// TwinCAT 3 PLC project Anthem
// ProgramVersion: 3.1.4023.0
// libraries:
//   Tc2_ModbusRTU, * (Beckhoff Automation GmbH)
//   Tc2_Standard, * (Beckhoff Automation GmbH)
//   Tc2_System, * (Beckhoff Automation GmbH)
//   Tc2_Utilities, * (Beckhoff Automation GmbH)
//   Tc3_Module, * (Beckhoff Automation GmbH)
// project tree:
//   / AnalogScaling.TcPOU, PlcTask.TcTTO
//   DUTs/ Block.TcDUT, EachRecipeStep.TcDUT, IndividualProcess.TcDUT, PhysicalIO.TcDUT, Properties.TcDUT, Pump.TcDUT, Reactor.TcDUT, Recipe.TcDUT, Valve.TcDUT, Vessel.TcDUT, VFD.TcDUT
//   GVLs/ IO.TcGVL, RecipeTags.TcGVL
//   Helpers/Assigner/ FB_Assigner.TcPOU, FB_TagAssignment.TcPOU, I_TagAssignment.TcIO
//   Helpers/ fbSimulator.TcPOU, FB_Scaling.TcPOU, MessageProvider.TcPOU, RecipeCommHandler.TcPOU
//   Helpers/RemainingTimeCalculator/ FBRemTimeCalc.TcPOU
//   Helpers/ShutDown/ FB_Shutdown.TcPOU, I_ShutDown.TcIO
//   Helpers/StirControl/ FbStirControl.TcPOU, IStirControl.TcIO
//   Helpers/VesselSelection/ FBSelection.TcPOU, ISelection.TcIO
//   ManualControl/ FB_ManualControl.TcPOU, I_ManualControl.TcIO
//   ManualControl/ManualImplementation/ FB_ManualImplementation.TcPOU, I_ManualImplementation.TcIO
//   Manualmplementation/ FB_ManualImplementation_1.TcPOU, I_ManualImplementation_1.TcIO
//   Manualmplementation/ManualControl/ FB_ManualControl_1.TcPOU, I_ManualControl_1.TcIO
//   POUs/ AnalogScaling_1.TcPOU, MAIN.TcPOU, Modbus.TcPOU
//   RecipeControl/ ClearRecipe.TcPOU, RecipeControl.TcPOU
//   RecipeControl/RecipeBlocks/Drain/ Drain.TcPOU
//   RecipeControl/RecipeBlocks/Flush/ FbFlush.TcPOU, IFlush.TcIO
//   RecipeControl/RecipeBlocks/N2Purge/ FbN2PurgeBlock.TcPOU, IN2PurgeBlock.TcIO, N2Purge.TcPOU
//   RecipeControl/RecipeBlocks/Stir/ FbStirBlock.TcPOU, IStirBlock.TcIO
//   RecipeControl/RecipeBlocks/Transfer/ ActivationLogic.TcPOU, EndLogic.TcPOU, Transfer.TcPOU
//   RecipeControl/RecipeBlocks/Wait/ fbWaitBlock.TcPOU, IWaitBlock.TcIO
// real-time tasks:
//   TASK PlcTask: cycle T#10ms, priority 20, ADS port 350

CONFIGURATION Anthem
    RESOURCE PLC ON TwinCAT3
        TASK PlcTask(INTERVAL := T#10ms, PRIORITY := 20);
        PROGRAM MAIN WITH PlcTask : MAIN;
    END_RESOURCE
END_CONFIGURATION

// ---- DUTs/Block.TcDUT
{attribute 'pack_mode' := '1'}
TYPE Block :
STRUCT
	Recipe 	: STRING(20);
	StepNo 	: DINT;
	Name 	: STRING(20);
	Properties : Properties;	

	
END_STRUCT
END_TYPE

// ---- DUTs/EachRecipeStep.TcDUT
TYPE EachRecipeStep :
STRUCT

   ///Tags for start block
    HeatCoolModeSelection:BOOL:=0; /// 0-is jacket mode/ 1-is process mode
	 HeatCoolDeltaTemp:DINT:=0; 
	 Started:BOOL:=0;
	 StartedTime:STRING:='';
	 Ended:BOOL:=0;
	 EndedTime:STRING:='';

	///Tags for HeatCoolBlock
	HeatCoolEnabled:BOOL:=0;
	HeatCoolStarted:BOOL:=0;
	HeatCoolStartedTime:STRING:='';
	HeatCoolEnded:BOOL:=0;
	HeatCoolEndedTime:STRING:='';
	HeatCoolSetPointExpression:DINT:=0;
	HeatCoolDuration:DINT:=0;
	HeatCoolOperatingMode:BOOL:=0;
	
	///Tags for StirrerBlock
	StirrerEnabled:BOOL:=0;
	StirrerStarted:BOOL:=0;
	StirrerStartedTime:STRING:='';
	StirrerEnded:BOOL:=0;
	StirrerEndedTime:STRING:='';
	StirrerSetPointExpression:DINT:=0;

	///Tags for DoseBlock	
	DosingEnabled:BOOL:=0;
	DosingStarted:BOOL:=0;
	DosingStartedTime:STRING:='';
	DosingEnded:BOOL:=0;
	DosingEndedTime:STRING:='';
    DosingMaxAmount:REAL:=0;
	DosingStopTemp:DINT:=0;
	DosingResumeTemp:DINT:=0;
	DosingRateSetpointExpression:REAL:=0;
	DosingMinRate:DINT:=0;
	DosingMaxRate:DINT:=0;
	DosingSettlingTime:DINT:=0;
	DosingMinPh:DINT:=0;
	DosingMaxPh:DINT:=0;
	DosingOperatingMode:BOOL:=0;
	
	////Tags for Wait tags
	WaitEnabled:BOOL:=0;
	WaitStarted:BOOL:=0;
	WaitStartedTime:STRING:='';
	WaitEndedTime:STRING:='';
	WaitEnded:BOOL:=0;
	WaitDuration:DINT:=0;
	WaitRemainingSeconds : INT;
	WaitRemainingMinutes : INT;
	WaitRemainingTime : STRING;
	
	//Tags for Centrifuge Block
	CentrifugeEnabled : BOOL;
	CentrifugeStarted : BOOL;
	CentrifugeEnded : BOOL;
	CentrifugeSpeedSetPoint : DINT;
	CentrifugeWaitTime : DINT;
	
	//Tags for Valves Block
	ValvesEnabled : BOOL;
	ValvesStarted : BOOL;
	ValvesEnded : BOOL;
	ValveAStatus : BOOL;
	ValveBStatus : BOOL;
	ValveCStatus : BOOL;
	
	//Tags for AOOD Pump Block
	AOODPumpEnabled : BOOL;
	AOODPumpStarted : BOOL;
	AOODPumpEnded : BOOL;
	Pump1Status : BOOL;
	Pump2Status : BOOL;

END_STRUCT
END_TYPE

// ---- DUTs/IndividualProcess.TcDUT
TYPE IndividualProcess :
STRUCT
	RawValue : INT;
	ScaledValue : LREAL;
	RawLowLimit : INT := 0;
	RawHighLimit : DINT := 32768;
	ScaledLowLimit : LREAL;
	ScaledHighLimit : LREAL;
END_STRUCT
END_TYPE

// ---- DUTs/PhysicalIO.TcDUT
TYPE PhysicalIO :
STRUCT
	R1_Valves AT %Q* : ARRAY[0..7] OF BOOL;
	R1_Pumps AT %Q* : ARRAY[0..1] OF BOOL;
	R1_LS AT %I* : ARRAY[0..1] OF BOOL;

	R2_Valves AT %Q* : ARRAY[0..7] OF BOOL;
	R2_Pumps AT %Q* : ARRAY[0..1] OF BOOL;
	R2_LS AT %I* : ARRAY[0..1] OF BOOL;

	R3_Valves AT %Q* : ARRAY[0..7] OF BOOL;
	R3_Pumps AT %Q* : ARRAY[0..1] OF BOOL;
	R3_LS AT %I* : ARRAY[0..1] OF BOOL;

	R4_Valves AT %Q* : ARRAY[0..7] OF BOOL;
	R4_Pumps AT %Q* : ARRAY[0..1] OF BOOL;
	R4_LS AT %I* : ARRAY[0..1] OF BOOL;

	R5_Valves AT %Q* : ARRAY[0..7] OF BOOL;
	R5_Pumps AT %Q* : ARRAY[0..1] OF BOOL;
	R5_LS AT %I* : ARRAY[0..1] OF BOOL;

	AA1_Valves AT %Q* : ARRAY[0..7] OF BOOL;
	AA1_Pumps AT %Q* : ARRAY[0..1] OF BOOL;
	AA1_LS AT %I* : ARRAY[0..1] OF BOOL;

	AA2_Valves AT %Q* : ARRAY[0..7] OF BOOL;
	AA2_Pumps AT %Q* : ARRAY[0..1] OF BOOL;
	AA2_LS AT %I* : ARRAY[0..1] OF BOOL;

	MVB_Valves AT %Q* : ARRAY[0..7] OF BOOL;
	MVB_Pumps AT %Q* : ARRAY[0..1] OF BOOL;
	MVB_LS AT %I* : ARRAY[0..1] OF BOOL;

	DCM_Valves AT %Q* : ARRAY[0..7] OF BOOL;
	DCM_Pumps AT %Q* : ARRAY[0..1] OF BOOL;
	DCM_LS AT %I* : ARRAY[0..1] OF BOOL;

	
	MVA_Valves AT %Q* : ARRAY[0..7] OF BOOL;
	MVA_Pumps AT %Q* : ARRAY[0..1] OF BOOL;
	MVA_AI AT %I* : ARRAY[0..4] OF INT;(*Temperature, Pressure, Level, VFD FB*)
	MVA_AO AT %Q* : ARRAY[0..1] OF INT;(*VFD*)
	
	RV50L_Valves AT %Q* : ARRAY[0..7] OF BOOL;
	RV50L_Pumps AT %Q* : ARRAY[0..1] OF BOOL;
	RV50L_AI AT %I* : ARRAY[0..4] OF INT;(*Temperature, Pressure, Level, VFD FB*)
	RV50L_AO AT %Q* : ARRAY[0..1] OF INT;(*VFD*)

	RV25L_Valves AT %Q* : ARRAY[0..7] OF BOOL;
	RV25L_Pumps AT %Q* : ARRAY[0..1] OF BOOL;
	RV25L_AI AT %I* : ARRAY[0..4] OF INT;(*Temperature, Pressure, Level, VFD FB*)
	RV25L_AO AT %Q* : ARRAY[0..1] OF INT;(*VFD*)
	
	SS_Tank AT %Q* : BOOL;
	DosingPumpEnable AT %Q* : BOOL;
	
	JacketTemperature AT %I* : INT;


END_STRUCT
END_TYPE

// ---- DUTs/Properties.TcDUT
{attribute 'pack_mode' := '1'}
TYPE Properties :
STRUCT
	bStartCommand : BOOL;
	bStopCommand : BOOL;
	bBlockStarted : BOOL;
	bBlockEnded : BOOL;
	sStartTime 	: STRING(10);
	sRemainingTime	: STRING(10);
	sEndTime	: STRING(10);
	sSource 	: STRING(20); (*Transfer blocks*)
	sDestination 	: STRING(20); (*Transfer blocks*)
	lrSetPoint 	: LREAL; (*Stirrer, HC blocks*)
	bModeSelection : BOOL; (*0=Jacket, 1=Process => HC Block and 0=Level, 1=Time => Transfer Block*)
	nInterval : DINT; (*Transfer, Wait Blocks*)
	sIntervalType : STRING(10); (*Seconds, Minutes, Hours => Wait, Transfer Blocks*)	


	
END_STRUCT
END_TYPE

// ---- DUTs/Pump.TcDUT
TYPE Pump EXTENDS Valve :
STRUCT
	nPulse : INT := 4;
	sTime : STRING;
	sRemainingTime : STRING;
END_STRUCT
END_TYPE

// ---- DUTs/Reactor.TcDUT
TYPE Reactor EXTENDS Vessel :
STRUCT
	Temperature : IndividualProcess;
	Pressure : IndividualProcess;
	Level : IndividualProcess;
	VFD : VFD;
END_STRUCT
END_TYPE

// ---- DUTs/Recipe.TcDUT
{attribute 'pack_mode' := '1'}
TYPE Recipe :
STRUCT
	Blocks : ARRAY[0..699] OF Block;
END_STRUCT
END_TYPE

// ---- DUTs/Valve.TcDUT
TYPE Valve :
STRUCT
	bStart : BOOL;
	Output : BOOL;
END_STRUCT
END_TYPE

// ---- DUTs/Vessel.TcDUT
TYPE Vessel :
STRUCT
	LLS : BOOL;	
	ULS : BOOL;	
	
	Valves : ARRAY[0..7] OF Valve;
	Pumps : ARRAY[0..1] OF Pump; 
//	VentValve : Valve;
//	N2PurgeValve : Valve;
//	TransferValve : Valve;
//	FillInValve : Valve;
//	FillInHeaderValve : Valve;
// 	DrainValve : Valve;
//	FlushingValve : Valve;

//	FillInPump : PUMP;
//	TransferPump : PUMP;
	
END_STRUCT
END_TYPE

// ---- DUTs/VFD.TcDUT
TYPE VFD :
STRUCT
	bStart : BOOL;
	bStop : BOOL;
	nRPMSetPointScaled : LREAL;
	nRPMFeedBackScaled : LREAL;
	nRPMFeedBackRaw : INT;
	nRPMSetPointRaw : INT;
END_STRUCT
END_TYPE

// ---- GVLs/IO.TcGVL
{attribute 'qualified_only'}
VAR_GLOBAL
	(*R 1..5, AA1, AA2, DCM, MVB*)
	Vessels : ARRAY[0..8] OF Vessel; 
	(* RV50L, RV25L, MVA  *)
	Reactors : ARRAY[0..2] OF Reactor;
	
	PhysicalIO : PhysicalIO;
	
	ChillerTempSetpoint : LREAL := 25;
	ChillerTemperature : LREAL;
	
	UpdateFieldPoint : INT;
	
	StirrerSetpoint_1 : REAL;
	
	JacketTemperature : LREAL;
	
	Temperature_1 : LREAL;
	Temperature_2 : LREAL;
	
	ReactorLevel_1 : int;
	ReactorLevel_2 : LREAL;

	Pressure_1 : LREAL;
	Pressure_2 : LREAL;

	StirrerCommand_1 : BOOL;
	StirrerCommand_2 : BOOL;
	
	HeatCoolFailure : BOOl;
	
END_VAR

// ---- GVLs/RecipeTags.TcGVL
{attribute 'qualified_only'}
VAR_GLOBAL
	SlaveRecipe : Recipe;
	Recipe	: Recipe;
	bRecipeStatus : BOOL;
	ClearRecipe : BOOL;
	bAbortRecipe : BOOL;
	bClearRecipe : BOOL;
	bPauseRecipe : BOOL;
	bResumeRecipe : BOOL;
	bSkipDrain : BOOL;
	bDrainStatus : BOOL;
	bRuntimeEdit : BOOL;
	CurrentExecutingStep: STRING;
	RecipeMessage: STRING;
	StaredTimeForRecipeBanner: STRING[255];
	
	bTransferStartTime : BOOL;
	
	bBlockEnd:ARRAY[0..699] OF BOOL;
	enWaitPause:ARRAY[0..699] OF BOOL;
	bBlockStart : ARRAY[0..699] OF BOOL;
	bStartTimeEnable : ARRAY[0..699] OF BOOL;

END_VAR

// ---- Helpers/Assigner/I_TagAssignment.TcIO
INTERFACE I_TagAssignment

METHOD AA1 : BOOL
VAR_INPUT
END_VAR
END_METHOD

METHOD AA2 : BOOL
VAR_INPUT
END_VAR
END_METHOD

METHOD DCM : BOOL
VAR_INPUT
END_VAR
END_METHOD

METHOD MVA : BOOL
VAR_INPUT
END_VAR
END_METHOD

METHOD MVB : BOOL
VAR_INPUT
END_VAR
END_METHOD

METHOD R1 : BOOL
VAR_INPUT
END_VAR
END_METHOD

METHOD R2 : BOOL
VAR_INPUT
END_VAR
END_METHOD

METHOD R3 : BOOL
VAR_INPUT
END_VAR
END_METHOD

METHOD R4 : BOOL
VAR_INPUT
END_VAR
END_METHOD

METHOD R5 : BOOL
VAR_INPUT
END_VAR
END_METHOD

METHOD RV : BOOL
VAR_INPUT
END_VAR
END_METHOD

END_INTERFACE

// ---- Helpers/ShutDown/I_ShutDown.TcIO

INTERFACE I_ShutDown

METHOD ShutDown : BOOL
VAR_INPUT
		GvlIdentifier : STRING;
END_VAR
END_METHOD

END_INTERFACE

// ---- Helpers/StirControl/IStirControl.TcIO
INTERFACE IStirControl

PROPERTY pSetpoint : LREAL
GET
END_GET
END_PROPERTY

METHOD StirControl : LREAL
VAR_INPUT
	i : INT;
END_VAR
END_METHOD

END_INTERFACE

// ---- Helpers/VesselSelection/ISelection.TcIO
INTERFACE ISelection

METHOD TargetConverter : INT
VAR_INPUT
	sTargetName : STRING;	
END_VAR
VAR_OUTPUT
	TargetConverter_output : INT;	
END_VAR
END_METHOD

END_INTERFACE

// ---- ManualControl/I_ManualControl.TcIO
INTERFACE I_ManualControl

METHOD M_RunPump : BOOL
VAR_INPUT
	bStart : BOOL;
	NTimes : INT;
END_VAR
END_METHOD

METHOD M_RunValve : BOOL
VAR_INPUT
	bStart : BOOL;
END_VAR
END_METHOD

END_INTERFACE

// ---- ManualControl/ManualImplementation/I_ManualImplementation.TcIO
INTERFACE I_ManualImplementation

PROPERTY ipManualControl : Array [0..12, 0..12] of I_ManualControl
GET
END_GET
END_PROPERTY

END_INTERFACE

// ---- Manualmplementation/I_ManualImplementation_1.TcIO
INTERFACE I_ManualImplementation_1

PROPERTY ipManualControl : Array [0..10, 0..10] of I_ManualControl
GET
END_GET
END_PROPERTY

END_INTERFACE

// ---- Manualmplementation/ManualControl/I_ManualControl_1.TcIO
INTERFACE I_ManualControl_1

METHOD M_RunPump : BOOL
VAR_INPUT
	bStart : BOOL;
	NTimes : INT;
END_VAR
END_METHOD

METHOD M_RunValve : BOOL
VAR_INPUT
	bStart : BOOL;
END_VAR
END_METHOD

END_INTERFACE

// ---- RecipeControl/RecipeBlocks/Flush/IFlush.TcIO
INTERFACE IFlush

METHOD Flush : BOOL
VAR_INPUT
END_VAR
END_METHOD

PROPERTY pEndFeedback : BOOL
GET
END_GET
END_PROPERTY

END_INTERFACE

// ---- RecipeControl/RecipeBlocks/N2Purge/IN2PurgeBlock.TcIO
INTERFACE IN2PurgeBlock

PROPERTY pEndFeedback : BOOL
GET
END_GET
END_PROPERTY

METHOD Purge : BOOL
VAR_INPUT
	bStartCommand : BOOL;
	sSourceName : STRING;
	nCurrentBlock : INT;	
END_VAR
END_METHOD

END_INTERFACE

// ---- RecipeControl/RecipeBlocks/Stir/IStirBlock.TcIO
INTERFACE IStirBlock

PROPERTY pEndFeedback : BOOL
GET
END_GET
END_PROPERTY

PROPERTY pStartFeedback : BOOL
GET
END_GET
END_PROPERTY

METHOD Stir : BOOL
VAR_INPUT
	sTargetName : STRING;
	bStirStartCommand : BOOL;
	bStirEndCommand : BOOL;
	nStirSetPoint : INT;
END_VAR
END_METHOD

END_INTERFACE

// ---- RecipeControl/RecipeBlocks/Wait/IWaitBlock.TcIO
INTERFACE IWaitBlock

END_INTERFACE

// ---- POUs/MAIN.TcPOU
PROGRAM MAIN
VAR
	
	fb_ManualControl : ARRAY[0..12, 0..12] OF FB_ManualControl;
	i_manualControl : ARRAY[0..12, 0..12] OF I_ManualControl;
	fb_ManualImplementation : FB_ManualImplementation;
	
	fb_ShutDown : FB_ShutDown;
	i_ShutDown : I_ShutDown;
	
	fb_TagAssignment : FB_TagAssignment;
	i_TagAssignment : I_TagAssignment;
	fb_Assigner : FB_Assigner;
	
	fbStirBlock : FbStirBlock;
	iStirBlock : IStirBlock;
	
	
	fbN2PurgeBlock : FbN2PurgeBlock;
	iN2PurgeBlock : IN2PurgeBlock;
	
	fbStirControl : FBStirControl;
	iStirControl : IStirControl;
	
	k: INT;
	k_1: INT;
	
	//fbJson 			: FB_JsonDomParser;
	jsonDoc 		: SJsonValue;
	jsonProp		: SJsonValue;
	jsonID 			: SJsonValue;
	jsonValue		: SJsonValue;
	//sMessage 		: STRING(255) := '{"Step":"1","Name":"Transfer","Value":"20"}';
	sMessageNested : STRING(255) := '{"Recipe": "01", "Step":"01", "Name":"Transfer", "Properties":
										{"Source":"R1", "Dest":"R2", "Mode": "TRUE", "nInterval":"30", "sIntervalType":"s"}}'; 
	currentStepNo: INT;
	
	fglocal : FB_LocalSystemTime;
	System_Time: TIMESTRUCT;
	currentHour : STRING;
	currentMinute : STRING;
	currentSecond : STRING;
	concatenatedHourMinuteString : STRING;
	
	sCurrentSecond : STRING;
	sCurrentHour : STRING;
	sCurrentMinute : STRING;
	sConcatenatedHourMinuteString : STRING;
	
	bRecipeLocalTimer: BOOL;
	nOfftimer: UDINT;
	TimeInSeconds: UDINT;
	
END_VAR



FOR k:= 0 TO 10 DO
	FOR k_1 := 0 TO 10 DO
		i_manualControl[k, k_1]:= fb_ManualControl[k, k_1];
	END_FOR
END_FOR

fb_ManualImplementation(i_ManualControl:= i_manualControl);

i_ShutDown := fb_ShutDown;
iStirBlock := fbStirBlock;
iN2PurgeBlock := fbN2PurgeBlock;
//fb_RecipeControl(ipshutDown := i_ShutDown, ipStirBlock := iStirBlock, ipTransfer := iTransfer);

fb_Assigner(i_TagAssignment := fb_TagAssignment);

RecipeControl.ipStirBlock := iStirBlock;
RecipeControl.ipN2PurgeBlock := iN2PurgeBlock;
RecipeControl();

//=========================================================
// Analog Scaling

AnalogScaling_1();


Modbus();


//=========================================================
// System Time

fglocal(
	sNetID:='',
	bEnable:=TRUE,
	dwCycle:=5,
	dwOpt:=1,
	tTimeOut:=DEFAULT_ADS_TIMEOUT,
	bValid=> ,
	systemTime=>System_Time ,
	tzID=> );
	
//update current hour and minute strings	
currentHour := WORD_TO_STRING(fglocal.systemTime.wHour);
currentMinute := WORD_TO_STRING(fglocal.systemTime.wMinute);
currentSecond := WORD_TO_STRING(fglocal.systemTime.wSecond);

concatenatedHourMinuteString := CONCAT(STR1:=currentHour, STR2:= ':');
concatenatedHourMinuteString := CONCAT(STR1:=concatenatedHourMinuteString, STR2:= currentMinute);


IF RecipeTags.bRecipeStatus THEN
	bRecipeLocalTimer := TRUE;	
ELSE
	bRecipeLocalTimer := FALSE;	
END_IF
IF bRecipeLocalTimer  THEN
	nOfftimer := nOfftimer + 1;
	
ELSE
	nOfftimer := 0; 
	TimeInSeconds := 0;
END_IF
IO.UpdateFieldPoint := STRING_TO_INT(currentSecond) MOD 60;

IF nOfftimer = 100 THEN
	TimeInSeconds := TimeInSeconds +1;	
	nOfftimer := 0;
END_IF



sCurrentSecond := LREAL_TO_STRING(TimeInSeconds MOD 60);
sCurrentMinute := INT_TO_STRING(ABS(LREAL_TO_INT(TimeInSeconds/60)));
sCurrentHour	:= 	INT_TO_STRING(ABS(LREAL_TO_INT(TimeInSeconds/3600)));
sConcatenatedHourMinuteString := CONCAT(STR1:=sCurrentHour, STR2:= ':');
sConcatenatedHourMinuteString := CONCAT(STR1:=sConcatenatedHourMinuteString, STR2:= sCurrentMinute);

END_PROGRAM

// ---- ManualControl/FB_ManualControl.TcPOU
FUNCTION_BLOCK FB_ManualControl IMPLEMENTS  I_ManualControl
VAR_INPUT
END_VAR
VAR_OUTPUT
END_VAR
VAR
	TEMP_1 : BOOL;
	Counter : INT;
	TEMP : BOOL;

	
END_VAR

{warning 'add method implementation '}
METHOD M_RunPump : BOOL
VAR_INPUT
	bStart	: BOOL;
	NTimes : INT;

END_VAR
VAR
	
END_VAR

IF NTimes <> 0 THEN
	IF TRUE THEN
	Counter := Counter + 1;
	END_IF
	IF Counter >= (100/(2*NTimes)) THEN
		TEMP := TRUE;
	ELSE
		TEMP := FALSE;
	END_IF
	IF Counter >= (200/(2*NTimes)) THEN
		Counter := 0;
	END_IF
ELSE
	RETURN;
END_IF

IF bstart THEN
	M_RunPump := TEMP;
ELSE
	M_RunPump := FALSE;
END_IF
END_METHOD

{warning 'add method implementation '}
METHOD M_RunValve : BOOL
VAR_INPUT
	bStart	: BOOL;
END_VAR
VAR
	
END_VAR
M_RunValve := bStart;
END_METHOD

END_FUNCTION_BLOCK

// ---- ManualControl/ManualImplementation/FB_ManualImplementation.TcPOU
FUNCTION_BLOCK FB_ManualImplementation IMPLEMENTS  I_ManualImplementation
VAR_INPUT
		i_ManualControl : ARRAY[0..12,0..12] OF I_ManualControl;
END_VAR
VAR_OUTPUT
END_VAR
VAR
	i: INT;
	j: INT;
	k: INT;
	k_1: INT;
	bDosingPumpEnableVessels: BOOL;
	bDosingPumpEnableReactors: BOOL;

END_VAR

//=========================================================
// Instantiation Logic


	FOR k:=0 TO 10 DO
		FOR k_1 := 0 TO 10 DO
			IF i_ManualControl[k, k_1] <> 0 THEN
			THIS^.i_ManualControl[k, k_1] := i_ManualControl[k, k_1];
		END_IF	
		END_FOR
		
	END_FOR


//=========================================================
// Count Declaration Logic

	

//=========================================================
// Manual Logic
	
	//Manual Logic for Vessels.Valves
	
	FOR i:=0 TO 8 DO
		FOR j :=0 TO 7 DO
			IO.Vessels[i].Valves[j].Output :=i_ManualControl[i, j].
				M_RunValve(IO.Vessels[i].Valves[j].bStart);
		END_FOR
	END_FOR
	
	//Manual Logic for Vessels.Pumps
	
	FOR i:=0 TO 8 DO
		FOR j :=0 TO 1 DO
			//IO.Vessels[i].Pumps[j].nPulse := 6;
			IO.Vessels[i].Pumps[j].Output :=i_ManualControl[i,j].
				M_RunPump(IO.Vessels[i].Pumps[j].bStart,IO.Vessels[i].Pumps[j].nPulse);
			IF IO.Vessels[i].Pumps[j].bStart THEN
				bDosingPumpEnableVessels := TRUE;
			ELSE
				bDosingPumpEnableVessels := FALSE;
			END_IF
		END_FOR
	END_FOR
	
	//Manual Logic for Reactors.Valves
	
	FOR i:=0 TO 1 DO
		FOR j :=0 TO 7 DO
			IO.Reactors[i].Valves[j].Output :=i_ManualControl[9+i,j].
				M_RunValve(IO.Reactors[i].Valves[j].bStart);
		END_FOR
	END_FOR
	
	//Manual Logic for Reactors.Pumps
	
	FOR i:=0 TO 1 DO
		FOR j :=0 TO 1 DO
			IO.Reactors[i].Pumps[j].nPulse := 4;
			IO.Reactors[i].Pumps[j].Output :=i_ManualControl[9+i,j+1].
				M_RunPump(IO.Reactors[i].Pumps[j].bStart,IO.Reactors[i].Pumps[j].nPulse);
			IF IO.Reactors[i].Pumps[j].bStart THEN
				bDosingPumpEnableReactors := TRUE;
			ELSE
				bDosingPumpEnableReactors := FALSE;
			END_IF
		END_FOR
	END_FOR
	

//=========================================================
// Dosing Pump Enable Logic

IF IO.Vessels[0].Pumps[0].bStart OR IO.Vessels[0].Pumps[1].bStart
	OR IO.Vessels[1].Pumps[0].bStart OR IO.Vessels[1].Pumps[1].bStart
	OR IO.Vessels[2].Pumps[0].bStart OR IO.Vessels[2].Pumps[1].bStart
	OR IO.Vessels[3].Pumps[0].bStart OR IO.Vessels[3].Pumps[1].bStart
	OR IO.Vessels[4].Pumps[0].bStart OR IO.Vessels[4].Pumps[1].bStart
	OR IO.Vessels[5].Pumps[0].bStart OR IO.Vessels[5].Pumps[1].bStart
	OR IO.Vessels[6].Pumps[0].bStart OR IO.Vessels[6].Pumps[1].bStart
	OR IO.Vessels[7].Pumps[0].bStart OR IO.Vessels[7].Pumps[1].bStart
	OR IO.Vessels[8].Pumps[0].bStart OR IO.Vessels[8].Pumps[1].bStart
	OR IO.Reactors[0].Pumps[0].bStart OR IO.Reactors[0].Pumps[1].bStart
	OR IO.Reactors[1].Pumps[0].bStart OR IO.Reactors[1].Pumps[1].bStart THEN
	IO.PhysicalIO.DosingPumpEnable := TRUE;
ELSE
	IO.PhysicalIO.DosingPumpEnable := FALSE;

END_IF

//IF bDosingPumpEnableVessels OR bDosingPumpEnableReactors THEN

//END_IF

PROPERTY ipManualControl : ARRAY [0..12,0..12] OF I_ManualControl
GET
ipManualControl	:= i_ManualControl;
END_GET
END_PROPERTY

END_FUNCTION_BLOCK

// ---- Helpers/ShutDown/FB_Shutdown.TcPOU
FUNCTION_BLOCK FB_Shutdown IMPLEMENTS I_ShutDown
VAR_INPUT
END_VAR
VAR_OUTPUT
END_VAR
VAR
END_VAR

{warning 'add method implementation '}
METHOD ShutDown : BOOL
VAR_INPUT
	GvlIdentifier	: STRING;
END_VAR
//IF GvlIdentifier = 'R1' THEN
//	R1.RecipeStatus		:= FALSE;
//	R1.HeatCoolStatus	:= FALSE;
//	R1.StirrerStatus	:= FALSE;
//	R1.AbortRecipe		:= FALSE;
//END_IF;
END_METHOD

END_FUNCTION_BLOCK

// ---- Helpers/Assigner/FB_TagAssignment.TcPOU
FUNCTION_BLOCK FB_TagAssignment IMPLEMENTS I_TagAssignment
VAR_INPUT
END_VAR
VAR_OUTPUT
END_VAR
VAR
END_VAR

METHOD AA1 : BOOL
IO.PhysicalIO.AA1_Valves[0] := IO.Vessels[5].Valves[0].Output;
IO.PhysicalIO.AA1_Valves[1] := IO.Vessels[5].Valves[1].Output;
IO.PhysicalIO.AA1_Valves[2] := IO.Vessels[5].Valves[2].Output;
IO.PhysicalIO.AA1_Valves[3] := IO.Vessels[5].Valves[3].Output;
IO.PhysicalIO.AA1_Valves[4] := IO.Vessels[5].Valves[4].Output;
IO.PhysicalIO.AA1_Valves[5] := IO.Vessels[5].Valves[5].Output;
IO.PhysicalIO.AA1_Valves[6] := IO.Vessels[5].Valves[6].Output;

IO.PhysicalIO.AA1_Pumps[0] := IO.Vessels[5].Pumps[0].Output;
IO.PhysicalIO.AA1_Pumps[1] := IO.Vessels[5].Pumps[1].Output;

IO.Vessels[5].ULS := NOT(IO.PhysicalIO.AA1_LS[1]);
IO.Vessels[5].LLS := IO.PhysicalIO.AA1_LS[0];

AA1 := TRUE;
END_METHOD

{warning 'add method implementation '}
METHOD AA2 : BOOL
IO.PhysicalIO.AA2_Valves[0] := IO.Vessels[6].Valves[0].Output;
IO.PhysicalIO.AA2_Valves[1] := IO.Vessels[6].Valves[1].Output;
IO.PhysicalIO.AA2_Valves[2] := IO.Vessels[6].Valves[2].Output;
IO.PhysicalIO.AA2_Valves[3] := IO.Vessels[6].Valves[3].Output;
IO.PhysicalIO.AA2_Valves[4] := IO.Vessels[6].Valves[4].Output;
IO.PhysicalIO.AA2_Valves[5] := IO.Vessels[6].Valves[5].Output;
IO.PhysicalIO.AA2_Valves[6] := IO.Vessels[6].Valves[6].Output;

IO.PhysicalIO.AA2_Pumps[0] := IO.Vessels[6].Pumps[0].Output;
IO.PhysicalIO.AA2_Pumps[1] := IO.Vessels[6].Pumps[1].Output;

IO.Vessels[6].ULS := NOT(IO.PhysicalIO.AA2_LS[1]);
IO.Vessels[6].LLS := IO.PhysicalIO.AA2_LS[0];


AA2 := TRUE;
END_METHOD

{warning 'add method implementation '}
METHOD DCM : BOOL
IO.PhysicalIO.DCM_Valves[0] := IO.Vessels[7].Valves[0].Output;
IO.PhysicalIO.DCM_Valves[1] := IO.Vessels[7].Valves[1].Output;
IO.PhysicalIO.DCM_Valves[2] := IO.Vessels[7].Valves[2].Output;
IO.PhysicalIO.DCM_Valves[3] := IO.Vessels[7].Valves[3].Output;
IO.PhysicalIO.DCM_Valves[4] := IO.Vessels[7].Valves[4].Output;
IO.PhysicalIO.DCM_Valves[5] := IO.Vessels[7].Valves[5].Output;
IO.PhysicalIO.DCM_Valves[6] := IO.Vessels[7].Valves[6].Output;

IO.PhysicalIO.DCM_Pumps[0] := IO.Vessels[7].Pumps[0].Output;
IO.PhysicalIO.DCM_Pumps[1] := IO.Vessels[7].Pumps[1].Output;

IO.Vessels[7].ULS := NOT(IO.PhysicalIO.DCM_LS[1]);
IO.Vessels[7].LLS := IO.PhysicalIO.DCM_LS[0];


DCM := TRUE;
END_METHOD

{warning 'add method implementation '}
METHOD MVA : BOOL
IO.PhysicalIO.MVA_Valves[0] := IO.Reactors[0].Valves[0].Output;
IO.PhysicalIO.MVA_Valves[1] := IO.Reactors[0].Valves[1].Output;
IO.PhysicalIO.MVA_Valves[2] := IO.Reactors[0].Valves[2].Output;
IO.PhysicalIO.MVA_Valves[3] := IO.Reactors[0].Valves[3].Output;
IO.PhysicalIO.MVA_Valves[4] := IO.Reactors[0].Valves[4].Output;
IO.PhysicalIO.MVA_Valves[5] := IO.Reactors[0].Valves[5].Output;
IO.PhysicalIO.MVA_Valves[6] := IO.Reactors[0].Valves[6].Output;
IO.PhysicalIO.MVA_Valves[7] := IO.Reactors[0].Valves[7].Output;



IO.PhysicalIO.MVA_Pumps[0] := IO.Reactors[0].Pumps[0].Output;
IO.PhysicalIO.MVA_Pumps[1] := IO.Reactors[0].Pumps[1].Output;

IO.Reactors[0].Temperature.RawValue := IO.PhysicalIO.MVA_AI[0];
IO.Reactors[0].Pressure.RawValue := IO.PhysicalIO.MVA_AI[1];
IO.Reactors[0].Level.RawValue := IO.PhysicalIO.MVA_AI[2];
IO.Reactors[0].VFD.nRPMFeedBackRaw := IO.PhysicalIO.MVA_AI[3];
IO.PhysicalIO.MVA_AO[0] := IO.Reactors[0].VFD.nRPMSetPointRaw;

IO.Reactors[0].Temperature.ScaledLowLimit := -90;
IO.Reactors[0].Temperature.ScaledHighLimit := 200;
IO.Reactors[0].Pressure.ScaledLowLimit := -1;
IO.Reactors[0].Pressure.ScaledHighLimit := 9;
IO.Reactors[0].Level.ScaledLowLimit := 100;
IO.Reactors[0].Level.ScaledHighLimit := 7;

MVA := TRUE;
END_METHOD

{warning 'add method implementation '}
METHOD MVB : BOOL
IO.PhysicalIO.MVB_Valves[0] := IO.Vessels[8].Valves[0].Output;
IO.PhysicalIO.MVB_Valves[1] := IO.Vessels[8].Valves[1].Output;
IO.PhysicalIO.MVB_Valves[2] := IO.Vessels[8].Valves[2].Output;
IO.PhysicalIO.MVB_Valves[3] := IO.Vessels[8].Valves[3].Output;
IO.PhysicalIO.MVB_Valves[4] := IO.Vessels[8].Valves[4].Output;
IO.PhysicalIO.MVB_Valves[5] := IO.Vessels[8].Valves[5].Output;
IO.PhysicalIO.MVB_Valves[6] := IO.Vessels[8].Valves[6].Output;

IO.PhysicalIO.MVB_Pumps[0] := IO.Vessels[8].Pumps[0].Output;
IO.PhysicalIO.MVB_Pumps[1] := IO.Vessels[8].Pumps[1].Output;

IO.Vessels[8].ULS := NOT(IO.PhysicalIO.MVB_LS[1]);
IO.Vessels[8].LLS := IO.PhysicalIO.MVB_LS[0];


MVB := TRUE;
END_METHOD

{warning 'add method implementation '}
METHOD R1 : BOOL
VAR
END_VAR
IO.PhysicalIO.R1_Valves[0] := IO.Vessels[0].Valves[0].Output;
IO.PhysicalIO.R1_Valves[1] := IO.Vessels[0].Valves[1].Output;
IO.PhysicalIO.R1_Valves[2] := IO.Vessels[0].Valves[2].Output;
IO.PhysicalIO.R1_Valves[3] := IO.Vessels[0].Valves[3].Output;
IO.PhysicalIO.R1_Valves[4] := IO.Vessels[0].Valves[4].Output;
IO.PhysicalIO.R1_Valves[5] := IO.Vessels[0].Valves[5].Output;
IO.PhysicalIO.R1_Valves[6] := IO.Vessels[0].Valves[6].Output;

IO.PhysicalIO.R1_Pumps[0] := IO.Vessels[0].Pumps[0].Output;
IO.PhysicalIO.R1_Pumps[1] := IO.Vessels[0].Pumps[1].Output;

IO.Vessels[0].ULS := NOT(IO.PhysicalIO.R1_LS[1]);
IO.Vessels[0].LLS := IO.PhysicalIO.R1_LS[0];

//R1 := TRUE;
END_METHOD

{warning 'add method implementation '}
METHOD R2 : BOOL
IO.PhysicalIO.R2_Valves[0] := IO.Vessels[1].Valves[0].Output;
IO.PhysicalIO.R2_Valves[1] := IO.Vessels[1].Valves[1].Output;
IO.PhysicalIO.R2_Valves[2] := IO.Vessels[1].Valves[2].Output;
IO.PhysicalIO.R2_Valves[3] := IO.Vessels[1].Valves[3].Output;
IO.PhysicalIO.R2_Valves[4] := IO.Vessels[1].Valves[4].Output;
IO.PhysicalIO.R2_Valves[5] := IO.Vessels[1].Valves[5].Output;
IO.PhysicalIO.R2_Valves[6] := IO.Vessels[1].Valves[6].Output;

IO.PhysicalIO.R2_Pumps[0] := IO.Vessels[1].Pumps[0].Output;
IO.PhysicalIO.R2_Pumps[1] := IO.Vessels[1].Pumps[1].Output;

IO.Vessels[1].ULS := NOT(IO.PhysicalIO.R2_LS[1]);
IO.Vessels[1].LLS := IO.PhysicalIO.R2_LS[0];


R2 := TRUE;
END_METHOD

{warning 'add method implementation '}
METHOD R3 : BOOL
IO.PhysicalIO.R3_Valves[0] := IO.Vessels[2].Valves[0].Output;
IO.PhysicalIO.R3_Valves[1] := IO.Vessels[2].Valves[1].Output;
IO.PhysicalIO.R3_Valves[2] := IO.Vessels[2].Valves[2].Output;
IO.PhysicalIO.R3_Valves[3] := IO.Vessels[2].Valves[3].Output;
IO.PhysicalIO.R3_Valves[4] := IO.Vessels[2].Valves[4].Output;
IO.PhysicalIO.R3_Valves[5] := IO.Vessels[2].Valves[5].Output;
IO.PhysicalIO.R3_Valves[6] := IO.Vessels[2].Valves[6].Output;

IO.PhysicalIO.R3_Pumps[0] := IO.Vessels[2].Pumps[0].Output;
IO.PhysicalIO.R3_Pumps[1] := IO.Vessels[2].Pumps[1].Output;

IO.Vessels[2].ULS := NOT(IO.PhysicalIO.R3_LS[1]);
IO.Vessels[2].LLS := IO.PhysicalIO.R3_LS[0];


R3 := TRUE;
END_METHOD

{warning 'add method implementation '}
METHOD R4 : BOOL
IO.PhysicalIO.R4_Valves[0] := IO.Vessels[3].Valves[0].Output;
IO.PhysicalIO.R4_Valves[1] := IO.Vessels[3].Valves[1].Output;
IO.PhysicalIO.R4_Valves[2] := IO.Vessels[3].Valves[2].Output;
IO.PhysicalIO.R4_Valves[3] := IO.Vessels[3].Valves[3].Output;
IO.PhysicalIO.R4_Valves[4] := IO.Vessels[3].Valves[4].Output;
IO.PhysicalIO.R4_Valves[5] := IO.Vessels[3].Valves[5].Output;
IO.PhysicalIO.R4_Valves[6] := IO.Vessels[3].Valves[6].Output;

IO.PhysicalIO.R4_Pumps[0] := IO.Vessels[3].Pumps[0].Output;
IO.PhysicalIO.R4_Pumps[1] := IO.Vessels[3].Pumps[1].Output;

IO.Vessels[3].ULS := NOT(IO.PhysicalIO.R4_LS[1]);
IO.Vessels[3].LLS := IO.PhysicalIO.R4_LS[0];


R4 := TRUE;
END_METHOD

{warning 'add method implementation '}
METHOD R5 : BOOL
IO.PhysicalIO.R5_Valves[0] := IO.Vessels[4].Valves[0].Output;
IO.PhysicalIO.R5_Valves[1] := IO.Vessels[4].Valves[1].Output;
IO.PhysicalIO.R5_Valves[2] := IO.Vessels[4].Valves[2].Output;
IO.PhysicalIO.R5_Valves[3] := IO.Vessels[4].Valves[3].Output;
IO.PhysicalIO.R5_Valves[4] := IO.Vessels[4].Valves[4].Output;
IO.PhysicalIO.R5_Valves[5] := IO.Vessels[4].Valves[5].Output;
IO.PhysicalIO.R5_Valves[6] := IO.Vessels[4].Valves[6].Output;

IO.PhysicalIO.R5_Pumps[0] := IO.Vessels[4].Pumps[0].Output;
IO.PhysicalIO.R5_Pumps[1] := IO.Vessels[4].Pumps[1].Output;

IO.Vessels[4].ULS := NOT(IO.PhysicalIO.R4_LS[1]);
IO.Vessels[4].LLS := IO.PhysicalIO.R4_LS[0];


R5 := TRUE;
END_METHOD

{warning 'add method implementation '}
METHOD RV : BOOL
IO.PhysicalIO.RV50L_Valves[0] := IO.Reactors[1].Valves[0].Output;
IO.PhysicalIO.RV50L_Valves[1] := IO.Reactors[1].Valves[1].Output;
IO.PhysicalIO.RV50L_Valves[2] := IO.Reactors[1].Valves[2].Output;
IO.PhysicalIO.RV50L_Valves[3] := IO.Reactors[1].Valves[3].Output;
IO.PhysicalIO.RV50L_Valves[4] := IO.Reactors[1].Valves[4].Output;
IO.PhysicalIO.RV50L_Valves[5] := IO.Reactors[1].Valves[5].Output;
IO.PhysicalIO.RV50L_Valves[6] := IO.Reactors[1].Valves[6].Output;
IO.PhysicalIO.RV50L_Valves[7] := IO.Reactors[1].Valves[7].Output;


IO.PhysicalIO.RV50L_Pumps[0] := IO.Reactors[1].Pumps[0].Output;
IO.PhysicalIO.RV50L_Pumps[1] := IO.Reactors[1].Pumps[1].Output;

IO.Reactors[1].Temperature.RawValue := IO.PhysicalIO.RV50L_AI[0];
IO.Reactors[1].Pressure.RawValue := IO.PhysicalIO.RV50L_AI[1];
IO.Reactors[1].Level.RawValue := IO.PhysicalIO.RV50L_AI[2];
IO.Reactors[1].VFD.nRPMFeedBackRaw := IO.PhysicalIO.RV50L_AI[3];
IO.PhysicalIO.RV50L_AO[0] := IO.Reactors[1].VFD.nRPMSetPointRaw;




IO.Reactors[1].Temperature.ScaledLowLimit := -90;
IO.Reactors[1].Temperature.ScaledHighLimit := 200;
IO.Reactors[1].Pressure.ScaledLowLimit := -1;
IO.Reactors[1].Pressure.ScaledHighLimit := 9;
IO.Reactors[1].Level.ScaledLowLimit := 100;
IO.Reactors[1].Level.ScaledHighLimit := 0;


IO.PhysicalIO.RV25L_Valves[0] := IO.Reactors[2].Valves[0].Output;
IO.PhysicalIO.RV25L_Valves[1] := IO.Reactors[2].Valves[1].Output;
IO.PhysicalIO.RV25L_Valves[2] := IO.Reactors[2].Valves[2].Output;
IO.PhysicalIO.RV25L_Valves[3] := IO.Reactors[2].Valves[3].Output;
IO.PhysicalIO.RV25L_Valves[4] := IO.Reactors[2].Valves[4].Output;
IO.PhysicalIO.RV25L_Valves[5] := IO.Reactors[2].Valves[5].Output;
IO.PhysicalIO.RV25L_Valves[6] := IO.Reactors[2].Valves[6].Output;
IO.PhysicalIO.RV25L_Valves[7] := IO.Reactors[2].Valves[7].Output;


IO.PhysicalIO.RV25L_Pumps[0] := IO.Reactors[2].Pumps[0].Output;
IO.PhysicalIO.RV25L_Pumps[1] := IO.Reactors[2].Pumps[1].Output;

IO.Reactors[2].Temperature.RawValue := IO.PhysicalIO.RV25L_AI[0];
IO.Reactors[2].Pressure.RawValue := IO.PhysicalIO.RV25L_AI[1];
IO.Reactors[2].Level.RawValue := IO.PhysicalIO.RV25L_AI[2];
IO.Reactors[2].VFD.nRPMFeedBackRaw := IO.PhysicalIO.RV25L_AI[3];
IO.PhysicalIO.RV25L_AO[0] := IO.Reactors[2].VFD.nRPMSetPointRaw;


IO.Reactors[2].Temperature.ScaledLowLimit := -90;
IO.Reactors[2].Temperature.ScaledHighLimit := 200;
IO.Reactors[2].Pressure.ScaledLowLimit := -1;
IO.Reactors[2].Pressure.ScaledHighLimit := 9;
IO.Reactors[2].Level.ScaledLowLimit := 100;
IO.Reactors[2].Level.ScaledHighLimit := 0;




RV := TRUE;
END_METHOD

END_FUNCTION_BLOCK

// ---- Helpers/Assigner/FB_Assigner.TcPOU
FUNCTION_BLOCK FB_Assigner
VAR_INPUT
	i_TagAssignment : I_TagAssignment;
END_VAR
VAR_OUTPUT
END_VAR
VAR
END_VAR

IF i_TagAssignment <> 0 THEN
		THIS^.i_TagAssignment := i_TagAssignment;
END_IF	
	


i_TagAssignment.R1();
i_TagAssignment.R2();
i_TagAssignment.R3();
i_TagAssignment.R4();
i_TagAssignment.R5();
i_TagAssignment.AA1();
i_TagAssignment.AA2();
i_TagAssignment.DCM();
i_TagAssignment.MVA();
i_TagAssignment.MVB();
i_TagAssignment.RV();

END_FUNCTION_BLOCK

// ---- RecipeControl/RecipeBlocks/Stir/FbStirBlock.TcPOU
FUNCTION_BLOCK FbStirBlock IMPLEMENTS IStirBlock
VAR_INPUT
	
END_VAR
VAR_OUTPUT
	bStirBlockStarted: BOOL;
	bStirBlockEnded: BOOL;
	
END_VAR
VAR
	FbSimulator : fbSimulator;
	CurrentTarget: INT;

END_VAR

{warning 'add property implementation'}
PROPERTY pEndFeedback : BOOL
GET
pEndFeedback := bStirBlockEnded;
END_GET
END_PROPERTY

{warning 'add property implementation'}
PROPERTY pStartFeedback : BOOL
GET
pStartFeedback := bStirBlockStarted;
END_GET
END_PROPERTY

{warning 'add method implementation '}
METHOD Stir : BOOL
VAR_INPUT
	sTargetName : STRING;
	bStirStartCommand : BOOL;
	bStirEndCommand : BOOL;
	nStirSetPoint : INT;
END_VAR
VAR
END_VAR
IF sTargetName = 'RV_50L' THEN
	CurrentTarget := 1;
ELSIF  sTargetName = 'RV_25L' THEN
	CurrentTarget := 2;	
ELSIF  sTargetName = 'MVA' THEN
	CurrentTarget := 0;	
END_IF

IF nStirSetPoint <> 0 AND RecipeTags.bRecipeStatus THEN


	IF bStirStartCommand AND NOT(bStirEndCommand)THEN
		bStirBlockStarted := TRUE;
		IO.Reactors[CurrentTarget].VFD.nRPMSetPointScaled := nStirSetPoint;
	ELSE
		bStirBlockStarted := FALSE;
		IO.Reactors[CurrentTarget].VFD.nRPMSetPointScaled := 0;
	END_IF
ELSE
	bStirBlockStarted := FALSE;
END_IF

IO.Reactors[CurrentTarget].VFD.bStart := bStirBlockStarted;

IO.Reactors[CurrentTarget].VFD.nRPMSetPointScaled := nStirSetPoint;
//FbSimulator(CurrentValue := IO.Reactors[CurrentTarget].VFD.nRPMFeedBackScaled, TargetValue :=  nStirSetPoint,SimulatedValue => IO.Reactors[CurrentTarget].VFD.nRPMFeedBackScaled );

//	IF R1.RecipeStep[R1.StepCount].StirrerStartedTime = '' THEN
//		R1.RecipeStep[R1.StepCount].StirrerStartedTime := Main.concatenatedHourMinuteString;
//	END_IF

IF ABS(IO.Reactors[CurrentTarget].VFD.nRPMFeedBackScaled - nStirSetPoint)<= 5 THEN
	bStirBlockEnded := TRUE;	
//	IF R1.RecipeStep[R1.StepCount].StirrerEndedTime = '' THEN
//			R1.RecipeStep[R1.StepCount].StirrerEndedTime := Main.concatenatedHourMinuteString;
//		END_IF
ELSE 
		bStirBlockEnded := FALSE;	

END_IF

Stir := true;
END_METHOD

END_FUNCTION_BLOCK

// ---- Helpers/fbSimulator.TcPOU
FUNCTION_BLOCK fbSimulator
VAR_INPUT
	CurrentValue : REAL;
	TargetValue : REAL;
END_VAR
VAR_OUTPUT
	SimulatedValue : REAL;
END_VAR
VAR
	random_value : LREAL;
	fb_ran : DRAND;
END_VAR

fb_ran(Seed := 0, Num => );
random_value := 0.1 * STRING_TO_REAL(LREAL_TO_FMTSTR(fb_ran.Num, 2, TRUE));
IF ABS(CurrentValue-TargetValue)>0.5 THEN
	IF CurrentValue < TargetValue THEN
		CurrentValue := CurrentValue + random_value;
	ELSE
		CurrentValue := CurrentValue - random_value;
	END_IF
END_IF
SimulatedValue := STRING_TO_REAL(LREAL_TO_FMTSTR(CurrentValue, 2, TRUE)); //Rounding again here to clear any errors above

END_FUNCTION_BLOCK

// ---- RecipeControl/RecipeBlocks/N2Purge/FbN2PurgeBlock.TcPOU
FUNCTION_BLOCK FbN2PurgeBlock IMPLEMENTS IN2PurgeBlock
VAR_INPUT
END_VAR
VAR_OUTPUT
	bN2PurgeBlockEnded: BOOL;

END_VAR
VAR
	fb_FTRIG : F_TRIG;
	fbSelection : FBSelection;
END_VAR

{warning 'add property implementation'}
PROPERTY pEndFeedback : BOOL
GET
pEndFeedback := bN2PurgeBlockEnded;
END_GET
END_PROPERTY

METHOD Purge : BOOL
VAR_INPUT
	bStartCommand : BOOL;
	sSourceName : STRING;
	nCurrentBlock : INT;	
END_VAR

VAR
	nSource: INT;
	b: BOOL;
	bN2PurgeStartTime: BOOL;
	nStartTimeInSeconds: INT;
	nTime: DINT;
	bPumpStart: BOOL;
	bRecipePause: BOOL;
	enWaitPause: BOOL;
	RemainingTime : DINT;
	SecondsToAddWhilePause : INT;
	tempSecondsToAddWhilePause: INT;
END_VAR
fbSelection.TargetConverter(sTargetName:= sSourceName, TargetConverter_output => nSource); 


bN2PurgeStartTime:=TRUE;
IF (bN2PurgeStartTime=TRUE) THEN
	RecipeTags.Recipe.Blocks[nCurrentBlock].Properties.sStartTime:=MAIN.sConcatenatedHourMinuteString;
	nStartTimeInSeconds := STRING_TO_INT(MAIN.sCurrentSecond);
	bN2PurgeStartTime :=  FALSE;
END_IF

IF RecipeTags.Recipe.Blocks[nCurrentBlock].Properties.sIntervalType = 'S' THEN
	nTime := RecipeTags.Recipe.Blocks[nCurrentBlock].Properties.nInterval;
ELSIF RecipeTags.Recipe.Blocks[nCurrentBlock].Properties.sIntervalType = 'M' THEN
	nTime := RecipeTags.Recipe.Blocks[nCurrentBlock].Properties.nInterval * 60;
ELSIF RecipeTags.Recipe.Blocks[nCurrentBlock].Properties.sIntervalType = 'H' THEN
	nTime := RecipeTags.Recipe.Blocks[nCurrentBlock].Properties.nInterval * 3600;
END_IF

IF enWaitPause THEN
	tempSecondsToAddWhilePause := tempSecondsToAddWhilePause + 1;
	SecondsToAddWhilePause := tempSecondsToAddWhilePause; 
ELSE
	tempSecondsToAddWhilePause := 0;
END_IF

//IF bStartCommand THEN
	
//END_IF
IF NOT(RecipeTags.bPauseRecipe) THEN
	enWaitPause := FALSE;
	bPumpStart := TRUE;
	RemainingTime := nTime- nStartTimeInSeconds-STRING_TO_DINT(MAIN.sCurrentSecond);
ELSE
	bPumpStart := FALSE;
	enWaitPause := TRUE;
END_IF

//IF  (nTime + nStartTimeInSeconds + TRUNC(SecondsToAddWhilePause/100)) <= (STRING_TO_INT(MAIN.sCurrentSecond)) THEN
IF  (nTime  + TRUNC(SecondsToAddWhilePause/100)) <= (STRING_TO_INT(MAIN.sCurrentSecond)) THEN
	RecipeTags.Recipe.Blocks[nCurrentBlock].Properties.bStopCommand := TRUE;
	RecipeTags.Recipe.Blocks[nCurrentBlock].Properties.sEndTime:=MAIN.sConcatenatedHourMinuteString;
	bPumpStart := FALSE;
END_IF

IF bPumpStart THEN
	IF nSource<9 THEN
		IO.Vessels[nSource].Valves[1].bStart := TRUE;
	END_IF
	IF nSource>=9 AND nSource<=11 THEN
		IO.Reactors[nSource-9].Valves[1].bStart := TRUE;
	END_IF
ELSE
	IF nSource<9 THEN
		IO.Vessels[nSource].Valves[1].bStart := FALSE;
	END_IF
	IF nSource>=9 AND nSource<=11 THEN
		IO.Reactors[nSource-9].Valves[1].bStart := FALSE;
	end_if
END_IF

fb_FTRIG(CLK:=bStartCommand, Q=> );

IF fb_FTRIG.Q THEN
	b := TRUE;
	bN2PurgeBlockEnded := TRUE;	
END_IF

//	bN2PurgeBlockEnded := TRUE;
END_METHOD

END_FUNCTION_BLOCK

// ---- Helpers/VesselSelection/FBSelection.TcPOU
FUNCTION_BLOCK FBSelection IMPLEMENTS ISelection
VAR_INPUT
END_VAR
VAR_OUTPUT
END_VAR
VAR
END_VAR

{warning 'add method implementation '}
METHOD TargetConverter : INT
VAR_INPUT
	sTargetName : STRING;	
END_VAR
VAR_OUTPUT
	TargetConverter_output : INT;	
END_VAR

VAR
	nTemp: INT;
	nVar: INT;
	bVar1: BOOL;
	bVar3: BOOL;
	bVar2: BOOL;
END_VAR
IF sTargetName = 'R1' THEN
	nTemp := 0;
ELSIF sTargetName = 'R2' THEN
	nTemp := 1;
ELSIF sTargetName = 'R3' THEN
	nTemp := 2;
ELSIF sTargetName = 'R4' THEN
	nTemp := 3;
ELSIF sTargetName = 'R5' THEN
	nTemp := 4;
ELSIF sTargetName = 'AA1' THEN
	nTemp := 5;
ELSIF sTargetName = 'AA2' THEN
	nTemp := 6;
ELSIF sTargetName = 'DCM' THEN
	nTemp := 7;
ELSIF sTargetName = 'MVB' THEN
	nTemp := 8;
ELSIF sTargetName = 'RV_50L' OR sTargetName = 'RV 50L' THEN
	nTemp := 10;
ELSIF sTargetName = 'MVA 25L' or sTargetName = 'MVA' THEN
	nTemp := 9;
ELSIF sTargetName = 'RV_25L' THEN
	nTemp := 11;
ELSIF sTargetName = 'Fill In' THEN
	nTemp := 12;
ELSIF sTargetName = 'Flash' THEN
	nTemp := 13;
ELSE
	nTemp := 14;	
END_IF

TargetConverter_output := nTemp;
END_METHOD

END_FUNCTION_BLOCK

// ---- Helpers/StirControl/FbStirControl.TcPOU
FUNCTION_BLOCK FbStirControl IMPLEMENTS IStirControl

VAR_OUTPUT
	VFDSetpointOutput : LREAL;
END_VAR
VAR
END_VAR

{warning 'add property implementation'}
PROPERTY pSetpoint : LREAL
GET
pSetpoint := VFDSetpointOutput;
END_GET
END_PROPERTY

{warning 'add method implementation '}
METHOD StirControl : LREAL
VAR_INPUT
	i : INT;
END_VAR

IF IO.Reactors[i].VFD.bStart THEN
	VFDSetpointOutput := IO.Reactors[i].VFD.nRPMSetPointScaled;
ELSE
	VFDSetpointOutput := 0;		
END_IF
END_METHOD

END_FUNCTION_BLOCK

// ---- RecipeControl/RecipeBlocks/Transfer/Transfer.TcPOU
PROGRAM Transfer
VAR
	nSource: INT;
	nDestination: INT;
	
	nStartTimeInSeconds :UDINT;
	nTime: UDINT;
	
	tempSecondsToAddWhilePause: DINT;
	SecondsToAddWhilePause: DINT;
	
	RemainingTime: UDINT;
	fbRTRIG: R_TRIG;
	fbRTRIGEnable : BOOL;
	fbRTRIG2: F_TRIG;
	fbRTRIG2Enable : BOOL;


	fbFTRIGLLS : F_TRIG;
	fbFTRIGLLSEnable : BOOL;
	fbFTRIGLLS2 : F_TRIG;
	fbFTRIGLLS2Enable : BOOL;
	fbFTRIGULS : F_TRIG;
	fbFTRIGULSEnable : BOOL;
	bCommandToPumpStart:BOOL;
	fbSelection : FBSelection;

	
	bStartCommand: BOOL;
	CLK: INT;
	Q: INT;
	btransferBlockEnded: BOOL;
	
	sSourceName: STRING;
	sDestinationName: STRING;
	bMode: BOOL;
	
	DestinationULSON: BOOL;
END_VAR

VAR_INPUT	
	nCurrentBlock : INT;
END_VAR

// RECEIVE SOURCE , DESTINATION AND MODE INFORMATION FROM THE BLOCK //

sSourceName:= RecipeTags.Recipe.Blocks[nCurrentBlock].Properties.sSource;
sDestinationName:=RecipeTags.Recipe.Blocks[nCurrentBlock].Properties.sDestination;
bMode := RecipeTags.Recipe.Blocks[nCurrentBlock].Properties.bModeSelection;

// Converting Names to NUmbers FROM HELPERS/VESSEL SELECTION.FBSELECTION.TARGETCONVERTER //

fbSelection.TargetConverter(sTargetName:= sSourceName, TargetConverter_output => nSource); 
fbSelection.TargetConverter(sTargetName:=sDestinationName, TargetConverter_output=>nDestination);






IF nSource<9 THEN
	fbFTRIGLLS(CLK:=IO.Vessels[nSource].LLS);
END_IF


IF nDestination<9 THEN
	DestinationULSON := Not(IO.Vessels[nDestination].ULS);

//ELSIF nDestination>=9 AND nDestination<=11 THEN
//	fbFTRIGLLS2(CLK:=IO.Vessels[nSource].LLS);
//	IF fbFTRIGLLS2.Q THEN
//		DestinationULSON := TRUE;
//	ELSE
//		DestinationULSON := FALSE;
//	END_IF
ELSE
	DestinationULSON :=  FALSE;
END_IF



IF fbFTRIGLLS.Q THEN
	fbFTRIGLLSEnable := TRUE;
END_IF


IF nSource=12 THEN
	fbRTRIG2(CLK:=IO.Vessels[nDestination].ULS);
END_IF



IF fbRTRIG2.Q THEN
	fbRTRIG2Enable := TRUE;
	RecipeTags.bBlockStart[nCurrentBlock] := FALSE;
END_IF	





// Start Time - Writing start time to structure //
IF RecipeTags.Recipe.Blocks[nCurrentBlock].Properties.sStartTime = '' THEN
	RecipeTags.StaredTimeForRecipeBanner := MAIN.concatenatedHourMinuteString;
END_IF
IF (RecipeTags.bTransferStartTime=FALSE) THEN
//	RecipeControl.StaredTimeForRecipeBanner := MAIN.concatenatedHourMinuteString;
	RecipeTags.Recipe.Blocks[nCurrentBlock].Properties.sStartTime:=MAIN.sConcatenatedHourMinuteString;
	nStartTimeInSeconds:= STRING_TO_UDINT(MAIN.sCurrentSecond);
	RecipeTags.bTransferStartTime:=  TRUE;
END_IF

// Time Intervals - Conversion of input time as per selection//

IF RecipeTags.Recipe.Blocks[nCurrentBlock].Properties.sIntervalType = 'S' THEN
	nTime := DINT_TO_UDINT(RecipeTags.Recipe.Blocks[nCurrentBlock].Properties.nInterval);
ELSIF RecipeTags.Recipe.Blocks[nCurrentBlock].Properties.sIntervalType = 'M' THEN
	nTime := DINT_TO_UDINT(RecipeTags.Recipe.Blocks[nCurrentBlock].Properties.nInterval * 60);
ELSIF RecipeTags.Recipe.Blocks[nCurrentBlock].Properties.sIntervalType = 'H' THEN
	nTime := DINT_TO_UDINT(RecipeTags.Recipe.Blocks[nCurrentBlock].Properties.nInterval * 3600);
END_IF

// Track time elapsed for resume when pause is released //

IF RecipeTags.enWaitPause[nCurrentBlock] THEN
	tempSecondsToAddWhilePause := tempSecondsToAddWhilePause + 1;
	SecondsToAddWhilePause := tempSecondsToAddWhilePause; 
ELSE
	tempSecondsToAddWhilePause := 0;
	SecondsToAddWhilePause :=0;
END_IF

// TO CHECK BLOCK START //

IF NOT(RecipeTags.bPauseRecipe) THEN
		RecipeTags.enWaitPause[nCurrentBlock] := FALSE;
		RecipeTags.bBlockStart[nCurrentBlock] := TRUE;
		//IF bmode THEN
		//	RemainingTime := ABS(nTime- nStartTimeInSeconds-STRING_TO_UDINT(MAIN.sCurrentSecond));
		//ELSE
		//	RemainingTime := 0;
		//END_IF
ELSE
		RecipeTags.bBlockStart[nCurrentBlock] := FALSE;
		RecipeTags.enWaitPause[nCurrentBlock] := TRUE;
END_IF

// TO CHECK BLOCK COMPLETION  //

IF bmode THEN
	// time based mode //
	IF  (nTime + nStartTimeInSeconds + DINT_TO_UDINT(TRUNC(SecondsToAddWhilePause/100))) 
		          <= (STRING_TO_UDINT(MAIN.sCurrentSecond)) OR DestinationULSON  OR fbRTRIG2Enable THEN
		RecipeTags.Recipe.Blocks[nCurrentBlock].Properties.bStopCommand := TRUE;
		RecipeTags.Recipe.Blocks[nCurrentBlock].Properties.sEndTime:=MAIN.sConcatenatedHourMinuteString;
		RecipeTags.bBlockStart[nCurrentBlock] := FALSE;
		RecipeTags.bBlockEnd[nCurrentBlock] := TRUE;
		fbFTRIGLLSEnable := FALSE;
		fbRTRIG2Enable := FALSE;
		
	ELSE
		RecipeTags.bBlockEnd[nCurrentBlock] := FALSE;
	END_IF
ELSE
	// level based mode //
	RecipeTags.bBlockEnd[nCurrentBlock] := FALSE;
	IF DestinationULSON OR fbRTRIG2Enable OR (fbFTRIGLLSEnable AND nDestination>=9 AND nDestination<12 ) THEN
		EndLogic(nCurrentBlock:=RecipeTags.bBlockEnd[nCurrentBlock]); 
		RecipeTags.bBlockEnd[nCurrentBlock] := TRUE;
		RecipeTags.bBlockStart[nCurrentBlock] := FALSE;
		fbFTRIGLLSEnable := FALSE;
		fbRTRIG2Enable := FALSE;
	END_IF
END_IF



ActivationLogic(nCurrentBlock:= nCurrentBlock, nSource:=nSource, nDestination:=nDestination);

   // IF BLOCK END HAS BEEN MADE TRUE //
EndLogic(nCurrentBlock:=RecipeTags.bBlockEnd[nCurrentBlock]);
IF EndLogic.OutputBool THEN
	fbRTRIGEnable := TRUE;
	RecipeTags.bBlockStart[nCurrentBlock] :=FALSE;
	EndLogic(nCurrentBlock:=RecipeTags.bBlockEnd[nCurrentBlock]);
END_IF

IF ((fbRTRIGEnable AND NOT(RecipeTags.bRuntimeEdit))  AND RecipeTags.Recipe.Blocks[nCurrentBlock].Name = 'Transfer') THEN
	ActivationLogic(nCurrentBlock:= nCurrentBlock, nSource:=nSource, nDestination:=nDestination);
	SecondsToAddWhilePause := 0;
	fbRTRIGEnable := FALSE;
	nTime := 0;
	RecipeTags.bTransferStartTime := FALSE;
	//nStartTimeInSeconds := 0;
	RecipeTags.bBlockStart[nCurrentBlock]  :=FALSE;
	RecipeTags.bStartTimeEnable[nCurrentBlock] := FALSE;
	RecipeTags.bBlockEnd[nCurrentBlock] := FALSE;
//	EndLogic(nCurrentBlock:=RecipeTags.bBlockEnd[nCurrentBlock]);
	RecipeTags.bStartTimeEnable[nCurrentBlock] :=  FALSE;
	RecipeTags.Recipe.Blocks[nCurrentBlock].Properties.sEndTime:=MAIN.sConcatenatedHourMinuteString;
	RecipeTags.Recipe.Blocks[nCurrentBlock].Properties.bStopCommand := TRUE;
	

END_IF

END_PROGRAM

// ---- RecipeControl/RecipeBlocks/Transfer/EndLogic.TcPOU
PROGRAM EndLogic
VAR
	fbRTRIG: R_TRIG;
	fbRTRIGFillInUpper : R_TRIG;
END_VAR
VAR_INPUT
//	In : INT;
	nCurrentBlock: BOOL;
END_VAR
VAR_OUTPUT
	OutputBool : BOOL;
END_VAR



fbRTRIG(CLK:=nCurrentBlock , Q=> ); 

OutputBool := fbRTRIG.Q;

END_PROGRAM

// ---- RecipeControl/RecipeBlocks/Transfer/ActivationLogic.TcPOU
PROGRAM ActivationLogic
VAR_INPUT
	nCurrentBlock: INT;
	nSource : INT;
	nDestination : INT;
END_VAR

//=========================================================
// Valve Logic
	
	//AND (nDestination <9)
	IF RecipeTags.bBlockStart[nCurrentBlock] THEN
		// All Vessels except aa1 and aa2Source
		IF nSource < 9 AND NOT(nSource = 5 OR nSource = 6 OR nSource=7) THEN
			IO.Vessels[nSource].Valves[0].bStart := TRUE;       // OPENING VENT VALVE //
			IO.Vessels[nSource].Valves[1].bStart := FALSE;      // CLOSING PURGE VALVE //  
			IF io.Vessels[nSource].LLS THEN                     // IF SOURCE LOWER LIQUID AVAILABLE //
				IO.Vessels[nSource].Valves[2].bStart := TRUE;     // OPEN TRANSFER VALVE //
			ELSE
				IO.Vessels[nSource].Valves[2].bStart := FALSE;    // CLOSE TRANSFER VALVE //
			END_IF
		END_IF
		
		// DCM Source to RV
		IF NOT(nSource<>7) AND nDestination=10 THEN
			IO.Vessels[nSource].Valves[0].bStart := TRUE;
			IO.Vessels[nSource].Valves[1].bStart := FALSE;
			IF io.Vessels[nSource].LLS THEN
				IO.Vessels[nSource].Valves[2].bStart := TRUE;
			ELSE
				IO.Vessels[nSource].Valves[2].bStart := FALSE;
			END_IF
		END_IF
		
		// DCM Source 
		IF NOT(nSource<>7) AND NOT(nDestination=10)THEN
			IO.Vessels[nSource].Valves[0].bStart := TRUE;
			IO.Vessels[nSource].Valves[1].bStart := FALSE;
			IF io.Vessels[nSource].LLS THEN
				IO.Vessels[nSource].Valves[6].bStart := TRUE;
			ELSE
				IO.Vessels[nSource].Valves[6].bStart := FALSE;
			END_IF
		END_IF
		
		// AA1 and AA2 with RV Source 
		IF (nSource = 5 OR nSource = 6) AND nDestination=10 THEN
			IO.Vessels[nSource].Valves[0].bStart := TRUE;
			IO.Vessels[nSource].Valves[1].bStart := FALSE;
			IF io.Vessels[nSource].LLS THEN
				IO.Vessels[nSource].Valves[5].bStart := TRUE;
			ELSE
				IO.Vessels[nSource].Valves[5].bStart := FALSE;
			END_IF
		END_IF
		
		// AA1 and AA2 with MVA Source 
		IF (nSource = 5 OR nSource = 6) AND nDestination=9 THEN
			IO.Vessels[nSource].Valves[0].bStart := TRUE;
			IO.Vessels[nSource].Valves[1].bStart := FALSE;
			IF io.Vessels[nSource].LLS THEN
				IO.Vessels[nSource].Valves[2].bStart := TRUE;
			ELSE
				IO.Vessels[nSource].Valves[2].bStart := FALSE;
			END_IF
		END_IF
		
		//R5 to MVB
		IF nDestination =8 AND nSource = 4 THEN
			IO.Vessels[nDestination].Valves[0].bStart := TRUE;
		END_IF
		
		//R1 to vessels
		IF nDestination <9 AND NOT(nSource = 12) AND nSource=0 THEN
			IO.Vessels[nDestination].Valves[0].bStart := TRUE;
			IO.Vessels[nDestination].Valves[1].bStart := FALSE;
			IF io.Vessels[nSource].LLS THEN
				IO.Vessels[nSource].Valves[4].bStart := TRUE;
				IO.Vessels[nDestination].Valves[4].bStart := TRUE;
			ELSE
				IO.Vessels[nSource].Valves[4].bStart := FALSE;
				IO.Vessels[nDestination].Valves[4].bStart := FALSE;
			END_IF
		END_IF
		
		//  Reactors to Vessels
		IF nSource >=9 AND NOT(nSource = 12) AND nDestination<9  THEN
			IO.Reactors[nSource-9].Valves[0].bStart := TRUE;
			IO.Reactors[nSource-9].Valves[1].bStart := FALSE;
			IO.Reactors[nSource-9].Valves[2].bStart := TRUE;
		END_IF
		
		// RV Destination
		IF nDestination >=10 AND NOT(nSource=0) AND nSource<9 THEN
			IO.Vessels[nSource].Valves[0].bStart := TRUE;

//			IF io.Vessels[nSource].LLS THEN
//			ELSE
//				IO.Vessels[nSource].Valves[0].bStart := FALSE;
//			END_IF
			IO.Reactors[nDestination-9].Valves[1].bStart := FALSE;
		END_IF
		
		//R1 to reactors 
		IF nSource=0 AND nDestination >=9 THEN
			IO.Reactors[nDestination-9].Valves[0].bStart := TRUE;
			IO.Reactors[nDestination-9].Valves[1].bStart := FALSE;
			IF io.Vessels[nSource].LLS THEN
				IF nDestination = 9 THEN
					IO.Reactors[nDestination-9].Valves[4].bStart := TRUE;
				ELSE 
					IO.Reactors[nDestination-9].Valves[4].bStart := TRUE;
				END_IF
//				IO.Vessels[nSource].Valves[4].bStart := TRUE;
			ELSE
//				IO.Vessels[nSource].Valves[4].bStart := FALSE;
				IO.Reactors[nDestination-9].Valves[4].bStart := FALSE;
				IO.Reactors[nDestination-9].Valves[4].bStart := FALSE;
			END_IF
		END_IF
		
		//R2-5,	AA1,2,MVB,DCM TO DCM,MVA,RV
		IF nDestination=9 OR nDestination =10 AND NOT(nSource=0) AND nSource<9 THEN
				//AND NOT(nSource = 5 OR nSource = 6) THEN
			IO.Reactors[nDestination-9].Valves[0].bStart := TRUE;
			IO.Reactors[nDestination-9].Valves[1].bStart := FALSE;
		END_IF
		
//		//R2-5,	AA1 TO MVB
//		IF nDestination =8  AND NOT(nSource=0) AND nSource<9 THEN
//				//AND NOT(nSource = 5 OR nSource = 6) THEN
//			IO.Reactors[nDestination-9].Valves[0].bStart := TRUE;
//			IO.Reactors[nDestination-9].Valves[1].bStart := FALSE;
//		END_IF
		
		//Filling OF VESSELS
		IF nSource = 12 AND NOT(nSource<12) AND nDestination<9 THEN
			IO.Vessels[nDestination].Valves[0].bStart := TRUE;
			IO.Vessels[nDestination].Valves[3].bStart := TRUE;
		END_IF
		
		//Flash
		IF nSource = 13 AND nDestination>=9 AND nDestination<11 THEN
			IO.Reactors[nDestination-9].Valves[0].bStart := TRUE;
			IO.Reactors[nDestination-9].Valves[6].bStart := TRUE;
			
			IF io.Vessels[0].LLS THEN             
				IO.Vessels[0].Valves[0].bStart := TRUE;	
				IO.Vessels[0].Valves[2].bStart := TRUE;
				IO.Vessels[0].Pumps[1].bStart := TRUE;
				IO.Vessels[0].Valves[0].bStart := TRUE;
			ELSE
					
				IO.Vessels[0].Valves[2].bStart := FALSE;
				IO.Vessels[0].Pumps[1].bStart := FALSE;
			END_IF
			
		END_IF
		
		//MVA to RV transer
		IF nSource =9 AND nDestination = 10 THEN
			IO.Reactors[nSource-9].Valves[0].bStart := TRUE;
			IO.Reactors[nSource-9].Valves[2].bStart := TRUE;
			IO.Reactors[nSource-9].Valves[7].bStart := TRUE;
			IO.Reactors[nDestination-9].Valves[0].bStart := TRUE;
		END_IF
		
	ELSE
		// DCM Source
		IF NOT(nSource<>7) THEN
			IO.Vessels[nSource].Valves[0].bStart := FALSE;
			IO.Vessels[nSource].Valves[1].bStart := FALSE;
			IO.Vessels[nSource].Valves[6].bStart := false;
		END_IF
		// DCM Source to RV
		IF NOT(nSource<>7) AND nDestination=10 THEN
			IO.Vessels[nSource].Valves[0].bStart := FALSE;
			IO.Vessels[nSource].Valves[1].bStart := FALSE;
			IO.Vessels[nSource].Valves[2].bStart := FALSE;
		END_IF
		IF nSource < 9 THEN
			IO.Vessels[nSource].Valves[0].bStart := FALSE;
			IO.Vessels[nSource].Valves[2].bStart := FALSE;
			IO.Vessels[nSource].Pumps[1].bStart := FALSE;
			//bCommandToPumpStart[0] := FALSE;
		END_IF
		
		// AA1 and AA2 Source
		IF nSource = 5 OR nSource = 6 THEN
			IO.Vessels[nSource].Valves[0].bStart := FALSE;
			IO.Vessels[nSource].Valves[1].bStart := FALSE;
			IO.Vessels[nSource].Valves[5].bStart := FALSE;
		END_IF
		
		// AA1 and AA2 with RV Source 
		IF nSource = 5 OR nSource = 6 AND nDestination=10 THEN
			IO.Vessels[nSource].Valves[0].bStart := FALSE;
			IO.Vessels[nSource].Valves[1].bStart := FALSE;
			IO.Vessels[nSource].Valves[5].bStart := FALSE;
		END_IF
		
		// AA1 and AA2 with MVA Source 
		IF nSource = 5 OR nSource = 6 AND nDestination=9 THEN
			IO.Vessels[nSource].Valves[0].bStart := FALSE;
			IO.Vessels[nSource].Valves[1].bStart := FALSE;
			IO.Vessels[nSource].Valves[6].bStart := FALSE;
		END_IF
		
		IF nDestination < 9 AND NOT(nSource = 12) THEN
			IO.Vessels[nSource].Pumps[1].bStart := false;
			IO.Vessels[nDestination].Valves[0].bStart := FALSE;
			IO.Vessels[nDestination].Valves[4].bStart := FALSE;
		END_IF
		IF nSource >=9 AND NOT(nSource = 12) THEN
			IO.Reactors[nSource-9].Valves[0].bStart := FALSE;
			IO.Reactors[nSource-9].Valves[2].bStart := FALSE;
		END_IF
		IF nDestination >=9 AND NOT(nSource=0) AND nSource<9  THEN
			IO.Reactors[nDestination-9].Valves[0].bStart := FALSE;
			IO.Reactors[nDestination-9].Valves[2].bStart := FALSE;
		END_IF
		IF nDestination >=9  THEN
			IO.Reactors[nDestination-9].Valves[0].bStart := FALSE;
			IO.Reactors[nDestination-9].Valves[4].bStart := FALSE;
		END_IF
		IF nSource = 12 AND NOT(nSource<12) AND nDestination<9 THEN
			IO.Vessels[nDestination].Valves[3].bStart := FALSE;
			IO.Vessels[nDestination].Valves[0].bStart := FALSE;

		END_IF
		IF nDestination =9 OR nDestination =10 AND NOT(nSource=0)  THEN
			IO.Reactors[nDestination-9].Valves[0].bStart := FALSE;
			IO.Reactors[nDestination-9].Valves[1].bStart := FALSE;
		END_IF
		//R5 to MVB
		IF nDestination =8 AND nSource = 4 THEN
			IO.Vessels[nDestination].Valves[0].bStart := FALSE;
		END_IF
		
		//Flush
		IF nSource = 13 AND nDestination>=9 AND nDestination<11 THEN
			IO.Reactors[nDestination-9].Valves[0].bStart := FALSE;
			IO.Reactors[nDestination-9].Valves[6].bStart := FALSE;
			
			IO.Vessels[0].Valves[0].bStart := FALSE;	
			IO.Vessels[0].Valves[2].bStart := FALSE;
			IO.Vessels[0].Pumps[1].bStart := FALSE;
		END_IF
		//MVA to RV transer
		IF nSource =9 AND nDestination = 10 THEN
			IO.Reactors[nSource-9].Valves[0].bStart := FALSE;
			IO.Reactors[nSource-9].Valves[2].bStart := FALSE;
			IO.Reactors[nSource-9].Valves[7].bStart := FALSE;
			IO.Reactors[nDestination-9].Valves[0].bStart := FALSE;
		END_IF
	END_IF


//=========================================================
// Pump Logic
	IF RecipeTags.bBlockStart[nCurrentBlock] THEN
		
		IF nSource < 9 AND NOT((nSource=5) OR (nSource=6))    THEN
			IF io.Vessels[nSource].LLS THEN                         // CHECK SOURCE LOWER//
				IO.Vessels[nSource].Pumps[1].bStart := TRUE;        // START PUMP // 
			ELSE
				IO.Vessels[nSource].Pumps[1].bStart := FALSE;       // STOP PUMP //
			END_IF
		END_IF
		IF nSource >= 9 AND NOT((nSource=12) OR (nSource=13)) THEN
				IO.Reactors[nSource-9].Pumps[1].bStart := TRUE;
		END_IF
		IF nSource = 12  THEN
			IF io.Vessels[nDestination].ULS THEN
				IO.Vessels[nDestination].Pumps[0].bStart := TRUE;
			ELSE
				IO.Vessels[nDestination].Pumps[0].bStart := FALSE;
			END_IF
			
		END_IF
		IF nSource = 13 THEN
			IF io.Vessels[0].LLS THEN
				IO.Vessels[0].Pumps[1].bStart := TRUE;
			END_IF
		END_IF
	ELSE
		IF nSource < 9  AND NOT((nSource=5) OR (nSource=6)) THEN
			IO.Vessels[nSource].Pumps[1].bStart := FALSE;
		END_IF
		IF nSource >= 9  THEN
				IO.Reactors[nSource-9].Pumps[1].bStart := FALSE;
		END_IF
		IF nSource = 12  THEN
			IO.Vessels[nDestination].Pumps[0].bStart := FALSE;
		END_IF
		IF nSource = 13 THEN
			IF io.Vessels[0].LLS THEN
				IO.Vessels[0].Pumps[1].bStart := FALSE;
			END_IF
		END_IF
	END_IF


//WHILE (IO.Vessels[nSource].LLS AND NOT(IO.Vessels[nDestination].ULS) AND bCommandToPumpStart[0]) DO
	//IO.Vessels[nSource].Pumps[1].bStart := TRUE;
//END_WHILE;

END_PROGRAM

// ---- RecipeControl/RecipeControl.TcPOU
PROGRAM RecipeControl
VAR_INPUT
	ipStirBlock : IStirBlock;
	ipN2PurgeBlock : IN2PurgeBlock;

END_VAR
VAR
	ipshutDown : I_Shutdown;
	CurrentCount: INT;
	nCurrentCount: INT;
	ctu: CTU;
	ctu_1: CTU;
	CurrentCount_1: INT;
	CU: INT;
	CV: INT;
	RESET: INT;
	PV: INT;
	nCurrentCount_1: INT;
	TotalStepsCount: INT;
	i: INT;
	nCurrentBlock: INT;
	sTemp: STRING(255);
	sTime : STRING(255);
	
	fbRTRIG : R_TRIG;
	fbFTRIG : F_TRIG;
	offtimer : ARRAY[0..700] OF INT;
	nTime : ARRAY[0..700] OF UDINT;
	bPumpStart : ARRAY[0..700] OF BOOL;
	bModeSelection: ARRAY[0..700] OF BOOL;
	bTransferEn: ARRAY[0..700] OF BOOL;
	bN2PurgeEn: BOOL;
	Temp: ARRAY[0..700] OF INT;
	fb_TOF: TOF;
	bTempBit: BOOL;
	fbRTRIG_1: R_TRIG;
	bWaitStartTime: BOOL;
	bN2PurgeStartTime: BOOL;
	nStartTimeInSeconds: ARRAY[0..699] OF UDINT;
	bTempStirrer: BOOL;


	TagToStoreCurrentStep: INT;
	bRecipePause: BOOL;
	RemainingTime: UDINT;
	enWaitBlock: BOOL;
	SecondsToAddWhilePause: INT;
	enWaitPause: BOOL;
	tempSecondsToAddWhilePause: INT;
	fb_FTRIG: F_TRIG;
	s1: STRING;
	s2: STRING;
	strRemainingTime: STRING(255);
	
	
	waitFBRemTimeCalc : FBRemTimeCalc;
	waitRemTime : STRING(255);
	
END_VAR

RecipeCommHandler();
MessageProvider();
//=========================================================
// Instantiation Logic


	IF ipshutDown <> 0 THEN
		ipshutDown := ipshutDown;
	END_IF
	
	IF ipStirBlock <> 0 THEN
		ipStirBlock := ipStirBlock;
	END_IF


//=========================================================
// Counter Check Logic

	ctu(
		CU:= IO.Reactors[0].Pumps[0].Output, 
		RESET:= , 
		PV:= , 
		Q=> , 
		CV=> CurrentCount);
		
	nCurrentCount := WORD_TO_INT(CurrentCount)/10;	
	
	ctu_1(
		CU:= IO.Reactors[1].Pumps[1].Output, 
		RESET:= , 
		PV:= , 
		Q=> , 
		CV=> CurrentCount_1);
	
	nCurrentCount_1 := WORD_TO_INT(CurrentCount_1)/10;	
	



//=========================================================
// Counter Logic

	TotalStepsCount:=0;
	FOR i := 0 TO 700 DO
		IF NOT(RecipeTags.Recipe.Blocks[i].StepNo = 0) THEN
			TotalStepsCount := TotalStepsCount + 1;
		END_IF
	END_FOR
	
	
	fbRTRIG_1(CLK := RecipeTags.bRecipeStatus, Q=> bTempBit);
	IF bTempBit = TRUE THEN
		RecipeTags.bPauseRecipe := FALSE;	
		RecipeTags.bAbortRecipe := FALSE;
		RecipeTags.Recipe.Blocks[0].Properties.bBlockStarted := TRUE;
		RecipeTags.Recipe.Blocks[1].Properties.bStartCommand := TRUE;
		RecipeTags.Recipe.Blocks[1].Properties.bBlockStarted := TRUE;
		RecipeTags.Recipe.Blocks[0].Properties.bStopCommand := TRUE;
		RecipeTags.Recipe.Blocks[0].Properties.sStartTime:=MAIN.sConcatenatedHourMinuteString;

		nCurrentBlock := 1;
		bWaitStartTime :=  TRUE;
		bN2PurgeStartTime := TRUE;
		bTempBit := FALSE;

	END_IF
	IF RecipeTags.bAbortRecipe OR RecipeTags.bClearRecipe THEN
		ClearRecipe();
		RecipeTags.bPauseRecipe := FALSE;	
		RecipeTags.bRecipeStatus := FALSE;
		RecipeTags.bClearRecipe := FALSE;
		nCurrentBlock := 0;
		RecipeTags.bAbortRecipe := FALSE;
		Temp[nCurrentBlock] := 0;
		FOR i := 0 TO 700 DO
			offtimer[i] := 0;
		END_FOR

	END_IF
	RecipeTags.CurrentExecutingStep := RecipeTags.Recipe.Blocks[nCurrentBlock].Name;
 	IF RecipeTags.Recipe.Blocks[nCurrentBlock].Properties.bStopCommand = TRUE AND NOT(RecipeTags.bAbortRecipe) THEN
			nCurrentBlock := nCurrentBlock+1;
			RecipeTags.Recipe.Blocks[nCurrentBlock].Properties.bBlockStarted := TRUE;
			RecipeTags.Recipe.Blocks[nCurrentBlock].Properties.bStartCommand := TRUE;

			RecipeTags.Recipe.Blocks[nCurrentBlock-1].Properties.bStartCommand := FALSE;
			RecipeTags.Recipe.Blocks[nCurrentBlock-1].Properties.bStopCommand := FALSE;
			RecipeTags.Recipe.Blocks[nCurrentBlock-1].Properties.bBlockEnded := TRUE;
			
	END_IF
	
//	FOR i := 1 TO (TotalStepsCount) DO
//		IF RecipeTags.Recipe.Blocks[i].Properties.bStopCommand = TRUE AND NOT(RecipeTags.bAbortRecipe) THEN
//			nCurrentBlock := nCurrentBlock+1;
//			RecipeTags.Recipe.Blocks[nCurrentBlock].Properties.bBlockStarted := TRUE;
//			RecipeTags.Recipe.Blocks[nCurrentBlock].Properties.bStartCommand := TRUE;

//			RecipeTags.Recipe.Blocks[i].Properties.bStartCommand := FALSE;
//			RecipeTags.Recipe.Blocks[i].Properties.bStopCommand := FALSE;
//			RecipeTags.Recipe.Blocks[i].Properties.bBlockEnded := TRUE;
			
//	END_IF
	
//	END_FOR

//=========================================================
// Pause Logic
	IF RecipeTags.bRecipeStatus AND NOT(RecipeTags.bPauseRecipe) THEN
		TagToStoreCurrentStep := nCurrentBlock;
		bRecipePause := FALSE;
	END_IF
	IF RecipeTags.bPauseRecipe AND RecipeTags.bRecipeStatus THEN
		bRecipePause := TRUE;
		FOR i:=0 TO 2 DO
			IO.Reactors[i].VFD.bStart := FALSE;
		END_FOR
	END_IF
	
	
//=========================================================
// Stir Logic

	
	IF RecipeTags.Recipe.Blocks[nCurrentBlock].Name = 'Stirrer' THEN
		IF RecipeTags.Recipe.Blocks[nCurrentBlock].Properties.bStartCommand= TRUE AND NOT(RecipeTags.bAbortRecipe)  THEN
			bTempStirrer := TRUE;
		ELSE
			bTempStirrer := FALSE;
		END_IF
		
		ipStirBlock.Stir(RecipeTags.Recipe.Blocks[nCurrentBlock].Properties.sDestination,
							RecipeTags.Recipe.Blocks[nCurrentBlock].Properties.bStartCommand, bRecipePause, LREAL_TO_INT(RecipeTags.Recipe.Blocks[nCurrentBlock].Properties.lrSetPoint));
		IF RecipeTags.Recipe.Blocks[nCurrentBlock].Properties.sStartTime = '' THEN
			RecipeTags.StaredTimeForRecipeBanner := MAIN.concatenatedHourMinuteString;
			RecipeTags.Recipe.Blocks[nCurrentBlock].Properties.sStartTime := MAIN.sConcatenatedHourMinuteString;
		END_IF
		
		IF ipStirBlock.pEndFeedback THEN
			RecipeTags.Recipe.Blocks[nCurrentBlock].Properties.sEndTime:=MAIN.sConcatenatedHourMinuteString;
		END_IF

		RecipeTags.Recipe.Blocks[nCurrentBlock].Properties.bStopCommand := ipStirBlock.pEndFeedback;
		
	END_IF
	

//=========================================================
// Transfer Logic
	IF RecipeTags.Recipe.Blocks[nCurrentBlock].Name = 'Transfer' THEN
		Transfer(nCurrentBlock:=nCurrentBlock);
	END_IF


	

//=========================================================
// N2 Purge Logic

	
	IF RecipeTags.Recipe.Blocks[nCurrentBlock].Name = 'N2Purge' THEN
		N2Purge(nCurrentBlock := nCurrentBlock, sSourceName := RecipeTags.Recipe.Blocks[nCurrentBlock].Properties.sSource );
	END_IF
	
	
//=========================================================
// Drain Logic

	
	IF RecipeTags.Recipe.Blocks[nCurrentBlock].Name = 'Drain' THEN
		Drain(nCurrentBlock := nCurrentBlock, sSourceName := RecipeTags.Recipe.Blocks[nCurrentBlock].Properties.sSource );
	END_IF
	
//=========================================================
// Wait Logic

	IF RecipeTags.Recipe.Blocks[nCurrentBlock].Name = 'Wait' THEN
		IF (bWaitStartTime=TRUE) THEN
			RecipeTags.Recipe.Blocks[nCurrentBlock].Properties.sStartTime:=MAIN.sConcatenatedHourMinuteString;
			nStartTimeInSeconds[nCurrentBlock] := STRING_TO_UDINT(MAIN.sCurrentSecond);
			bWaitStartTime :=  FALSE;
		END_IF
		IF enWaitPause THEN
			tempSecondsToAddWhilePause := tempSecondsToAddWhilePause + 1;
			SecondsToAddWhilePause := tempSecondsToAddWhilePause; 
		ELSE
			tempSecondsToAddWhilePause := 0;
		END_IF
		
		IF RecipeTags.Recipe.Blocks[nCurrentBlock].Properties.sIntervalType = 'S' THEN
				nTime[nCurrentBlock] := DINT_TO_UDINT(RecipeTags.Recipe.Blocks[nCurrentBlock].Properties.nInterval);
		ELSIF RecipeTags.Recipe.Blocks[nCurrentBlock].Properties.sIntervalType = 'M' THEN
				nTime[nCurrentBlock] := DINT_TO_UDINT(RecipeTags.Recipe.Blocks[nCurrentBlock].Properties.nInterval * 60);
		ELSIF RecipeTags.Recipe.Blocks[nCurrentBlock].Properties.sIntervalType = 'H' THEN
				nTime[nCurrentBlock] := DINT_TO_UDINT(RecipeTags.Recipe.Blocks[nCurrentBlock].Properties.nInterval * 3600);
		END_IF
		IF RecipeTags.Recipe.Blocks[nCurrentBlock].Properties.bBlockStarted = TRUE THEN
			IF NOT(bRecipePause) THEN
				enWaitPause := FALSE;
				RemainingTime := ABS(nTime[nCurrentBlock]- nStartTimeInSeconds[nCurrentBlock]-STRING_TO_UDINT(MAIN.sCurrentSecond));
				
				
				RecipeTags.Recipe.Blocks[nCurrentBlock].Properties.sRemainingTime := waitRemTime;
				IF (nTime[nCurrentBlock] + nStartTimeInSeconds[nCurrentBlock] + TRUNC(SecondsToAddWhilePause/100)) = (STRING_TO_INT(MAIN.sCurrentSecond)) THEN
					bWaitStartTime := TRUE;
					RemainingTime := 0;
					RecipeTags.Recipe.Blocks[nCurrentBlock].Properties.sEndTime:=MAIN.sConcatenatedHourMinuteString;
					RecipeTags.Recipe.Blocks[nCurrentBlock].Properties.bStopCommand := TRUE;

				END_IF
			ELSE
				enWaitPause := True;

			END_IF
			
		END_IF
		
	END_IF

	waitFBRemTimeCalc(udRemainingTime:=RemainingTime);
				
	waitRemTime := waitFBRemTimeCalc.strRemainingTime;
//=========================================================
// End Logic

	
	IF RecipeTags.Recipe.Blocks[nCurrentBlock].Name = 'End' THEN
		RecipeTags.Recipe.Blocks[nCurrentBlock].Properties.bBlockStarted := TRUE;
		RecipeTags.Recipe.Blocks[nCurrentBlock].Properties.sEndTime:=MAIN.sConcatenatedHourMinuteString;
		FOR i:=0 TO 2 DO
			IO.Reactors[i].VFD.bStart := FALSE;
			IO.Reactors[i].VFD.nRPMSetPointScaled :=0;
		END_FOR
		RecipeTags.bRecipeStatus := FALSE;
		RecipeTags.Recipe.Blocks[nCurrentBlock].Properties.bBlockEnded := TRUE;
	END_IF

END_PROGRAM

// ---- Helpers/RemainingTimeCalculator/FBRemTimeCalc.TcPOU
FUNCTION_BLOCK FBRemTimeCalc
VAR_INPUT
	udRemainingTime: UDINT;
END_VAR
VAR_OUTPUT
	strRemainingTime: STRING(255);
END_VAR
VAR
	s1: STRING(255);
	s2: STRING(255);
END_VAR

s1 := INT_TO_STRING(REAL_TO_INT(udRemainingTime/60));
s2 := INT_TO_STRING(REAL_TO_INT(udRemainingTime MOD 60));
				
IF STRING_TO_INT(s1) < 10 THEN
	s1 := concat('0',s1);
ELSE
	s1 := s1;
END_IF
IF STRING_TO_INT(s2) < 10 THEN
	s2 := concat('0',s2);
ELSE
	s2 := s2;
END_IF
				
strRemainingTime := concat(s1, concat(':',s2));

END_FUNCTION_BLOCK

// ---- Helpers/RecipeCommHandler.TcPOU
PROGRAM RecipeCommHandler
VAR
	i: INT;
	RuntimeEdit : F_TRIG;
	FinalUpdate : F_TRIG;

	bRuntimeEditDone: BOOL;
	bFinalUpdateAfterEndBlock : BOOL;
END_VAR

RuntimeEdit(CLK:=RecipeTags.bRuntimeEdit);

IF RuntimeEdit.Q THEN
	bRuntimeEditDone := TRUE;
END_IF
//OnRecipeTriggerEdit(CLK:=RecipeTags.bRecipeStatus);




IF RecipeTags.bRecipeStatus AND NOT(RecipeTags.bRuntimeEdit) AND NOT(bRuntimeEditDone) THEN
//IF RecipeTags.bRecipeStatus  THEN
	FOR i := 0 TO 699 DO
		RecipeTags.Recipe.Blocks[i].Name := Recipetags.SlaveRecipe.Blocks[i].Name;
		RecipeTags.Recipe.Blocks[i].StepNo := Recipetags.SlaveRecipe.Blocks[i].StepNo;
		RecipeTags.Recipe.Blocks[i].Properties.sSource := Recipetags.SlaveRecipe.Blocks[i].Properties.sSource;
		RecipeTags.Recipe.Blocks[i].Properties.sDestination := Recipetags.SlaveRecipe.Blocks[i].Properties.sDestination;
		RecipeTags.Recipe.Blocks[i].Properties.bModeSelection := Recipetags.SlaveRecipe.Blocks[i].Properties.bModeSelection;
		RecipeTags.Recipe.Blocks[i].Properties.lrSetPoint := Recipetags.SlaveRecipe.Blocks[i].Properties.lrSetPoint;
		RecipeTags.Recipe.Blocks[i].Properties.nInterval := Recipetags.SlaveRecipe.Blocks[i].Properties.nInterval;
		RecipeTags.Recipe.Blocks[i].Properties.sIntervalType := Recipetags.SlaveRecipe.Blocks[i].Properties.sIntervalType;
	END_FOR
	FOR i := 0 TO 699 DO
		RecipeTags.SlaveRecipe.Blocks[i].Properties.bBlockEnded := Recipetags.Recipe.Blocks[i].Properties.bBlockEnded;
		RecipeTags.SlaveRecipe.Blocks[i].Properties.bBlockStarted := Recipetags.Recipe.Blocks[i].Properties.bBlockStarted;
		RecipeTags.SlaveRecipe.Blocks[i].Properties.bStartCommand := Recipetags.Recipe.Blocks[i].Properties.bStartCommand;
		RecipeTags.SlaveRecipe.Blocks[i].Properties.bStopCommand := Recipetags.Recipe.Blocks[i].Properties.bStopCommand;
		RecipeTags.SlaveRecipe.Blocks[i].Properties.sStartTime := Recipetags.Recipe.Blocks[i].Properties.sStartTime;
		RecipeTags.SlaveRecipe.Blocks[i].Properties.sEndTime := Recipetags.Recipe.Blocks[i].Properties.sEndTime;
		RecipeTags.SlaveRecipe.Blocks[i].Properties.sRemainingTime := Recipetags.Recipe.Blocks[i].Properties.sRemainingTime;

	END_FOR
END_IF
IF bRuntimeEditDone THEN
	FOR i := RecipeControl.nCurrentBlock TO RecipeControl.TotalStepsCount DO
		RecipeTags.Recipe.Blocks[i].Name := Recipetags.SlaveRecipe.Blocks[i].Name;
		RecipeTags.Recipe.Blocks[i].StepNo := Recipetags.SlaveRecipe.Blocks[i].StepNo;
		RecipeTags.Recipe.Blocks[i].Properties.sSource := Recipetags.SlaveRecipe.Blocks[i].Properties.sSource;
		RecipeTags.Recipe.Blocks[i].Properties.sDestination := Recipetags.SlaveRecipe.Blocks[i].Properties.sDestination;
		RecipeTags.Recipe.Blocks[i].Properties.bModeSelection := Recipetags.SlaveRecipe.Blocks[i].Properties.bModeSelection;
		RecipeTags.Recipe.Blocks[i].Properties.lrSetPoint := Recipetags.SlaveRecipe.Blocks[i].Properties.lrSetPoint;
		RecipeTags.Recipe.Blocks[i].Properties.nInterval := Recipetags.SlaveRecipe.Blocks[i].Properties.nInterval;
		RecipeTags.Recipe.Blocks[i].Properties.sIntervalType := Recipetags.SlaveRecipe.Blocks[i].Properties.sIntervalType;
	END_FOR
	FOR i := 0 TO RecipeControl.nCurrentBlock DO
		RecipeTags.SlaveRecipe.Blocks[i].Name := Recipetags.Recipe.Blocks[i].Name;
		RecipeTags.SlaveRecipe.Blocks[i].StepNo := Recipetags.Recipe.Blocks[i].StepNo;
		RecipeTags.SlaveRecipe.Blocks[i].Properties.bBlockStarted := RecipeTags.Recipe.Blocks[i].Properties.bBlockStarted;
		RecipeTags.SlaveRecipe.Blocks[i].Properties.bBlockEnded := Recipetags.Recipe.Blocks[i].Properties.bBlockEnded;
		RecipeTags.SlaveRecipe.Blocks[i].Properties.bStartCommand := Recipetags.Recipe.Blocks[i].Properties.bStartCommand;
		RecipeTags.SlaveRecipe.Blocks[i].Properties.bStopCommand := Recipetags.Recipe.Blocks[i].Properties.bStopCommand;
		RecipeTags.SlaveRecipe.Blocks[i].Properties.sStartTime := Recipetags.Recipe.Blocks[i].Properties.sStartTime;
		RecipeTags.SlaveRecipe.Blocks[i].Properties.sEndTime := Recipetags.Recipe.Blocks[i].Properties.sEndTime;
		RecipeTags.SlaveRecipe.Blocks[i].Properties.sRemainingTime := Recipetags.Recipe.Blocks[i].Properties.sRemainingTime;
	END_FOR
	bRuntimeEditDone := FALSE;
END_IF
//To Handle the situation where the recipestatus turning off as soon as the end block completed
FinalUpdate(CLK:=Recipetags.bRecipeStatus);

IF FinalUpdate.Q THEN
	bFinalUpdateAfterEndBlock := TRUE;
END_IF


IF bFinalUpdateAfterEndBlock THEN
	FOR i := 0 TO 699 DO
		RecipeTags.SlaveRecipe.Blocks[i].Properties.bBlockEnded := Recipetags.Recipe.Blocks[i].Properties.bBlockEnded;
		RecipeTags.SlaveRecipe.Blocks[i].Properties.bBlockStarted := Recipetags.Recipe.Blocks[i].Properties.bBlockStarted;
	END_FOR
	bFinalUpdateAfterEndBlock := false;
END_IF

END_PROGRAM

// ---- Helpers/MessageProvider.TcPOU
PROGRAM MessageProvider
VAR
	Message : ARRAY[0..10] OF STRING;
	FinalMessage : STRING[1000];
	i: INT;
END_VAR



IF RecipeTags.Recipe.Blocks[RecipeControl.nCurrentBlock].Properties.bBlockStarted AND RecipeTags.Recipe.Blocks[RecipeControl.nCurrentBlock].Name='Transfer' THEN
	Message[0] := concat(RecipeTags.Recipe.Blocks[RecipeControl.nCurrentBlock].Name,' - ');
	Message[1] := concat(Message[0], RecipeTags.Recipe.Blocks[RecipeControl.nCurrentBlock].Properties.sSource );
	Message[2] := concat(Message[1],' to ' );
	Message[3] := concat(Message[2], RecipeTags.Recipe.Blocks[RecipeControl.nCurrentBlock].Properties.sDestination);
	Message[4] := concat(Message[3], ' Started At ');
	Message[5] := concat(Message[4], RecipeTags.StaredTimeForRecipeBanner);
	RecipeTags.RecipeMessage := Message[5];
END_IF


IF RecipeTags.Recipe.Blocks[RecipeControl.nCurrentBlock].Properties.bBlockStarted AND RecipeTags.Recipe.Blocks[RecipeControl.nCurrentBlock].Name='Stirrer' THEN
	Message[0] := concat(RecipeTags.Recipe.Blocks[RecipeControl.nCurrentBlock].Name,' - ');
	Message[1] := concat(Message[0], RecipeTags.Recipe.Blocks[RecipeControl.nCurrentBlock].Properties.sSource );
	Message[2] := concat(Message[1], ' Started At ');
	Message[3] := concat(Message[2], RecipeTags.StaredTimeForRecipeBanner);
	RecipeTags.RecipeMessage := Message[3];
END_IF

IF RecipeTags.Recipe.Blocks[RecipeControl.nCurrentBlock].Properties.bBlockStarted AND RecipeTags.Recipe.Blocks[RecipeControl.nCurrentBlock].Name='Drain' THEN
	Message[0] := concat(RecipeTags.Recipe.Blocks[RecipeControl.nCurrentBlock].Name,' - ');
	Message[1] := concat(Message[0], RecipeTags.Recipe.Blocks[RecipeControl.nCurrentBlock].Properties.sSource );
	Message[2] := concat(Message[1], ' Started At ');
	Message[3] := concat(Message[2], RecipeTags.StaredTimeForRecipeBanner);
	RecipeTags.RecipeMessage := Message[3];
END_IF


IF RecipeTags.Recipe.Blocks[RecipeControl.nCurrentBlock].Properties.bBlockStarted AND RecipeTags.Recipe.Blocks[RecipeControl.nCurrentBlock].Name='N2Purge' THEN
	Message[0] := concat(RecipeTags.Recipe.Blocks[RecipeControl.nCurrentBlock].Name,' - ');
	Message[1] := concat(Message[0], RecipeTags.Recipe.Blocks[RecipeControl.nCurrentBlock].Properties.sSource );
	Message[2] := concat(Message[1], ' Started At ');
	Message[3] := concat(Message[2], RecipeTags.StaredTimeForRecipeBanner);
	RecipeTags.RecipeMessage := Message[3];
END_IF


IF RecipeTags.Recipe.Blocks[RecipeControl.nCurrentBlock].Properties.bBlockStarted AND RecipeTags.Recipe.Blocks[RecipeControl.nCurrentBlock].Name='Wait' THEN
	Message[0] := concat(RecipeTags.Recipe.Blocks[RecipeControl.nCurrentBlock].Name,' - ');
	Message[1] := concat(Message[0], RecipeTags.Recipe.Blocks[RecipeControl.nCurrentBlock].Properties.sSource );
	Message[2] := concat(Message[1], ' Started At ');
	Message[3] := concat(Message[2], RecipeTags.StaredTimeForRecipeBanner);
	RecipeTags.RecipeMessage := Message[3];
END_IF

IF RecipeTags.Recipe.Blocks[RecipeControl.nCurrentBlock].Properties.bBlockStarted AND RecipeTags.Recipe.Blocks[RecipeControl.nCurrentBlock].Name='Start' THEN
	Message[0] := concat('Recipe Started At ',RecipeTags.StaredTimeForRecipeBanner);
	RecipeTags.RecipeMessage := Message[0];
END_IF


IF RecipeTags.Recipe.Blocks[RecipeControl.nCurrentBlock].Properties.bBlockStarted AND RecipeTags.Recipe.Blocks[RecipeControl.nCurrentBlock].Name='End' THEN
	Message[0] := concat('Recipe Ended At ',RecipeTags.StaredTimeForRecipeBanner);
	RecipeTags.RecipeMessage := Message[0];
END_IF

IF RecipeTags.Recipe.Blocks[RecipeControl.nCurrentBlock].Name='' THEN
	
	FOR i:=0 TO 10 DO
		Message[i] := ''; 
	END_FOR
	RecipeTags.RecipeMessage := '';
END_IF

END_PROGRAM

// ---- RecipeControl/RecipeBlocks/Drain/Drain.TcPOU
PROGRAM Drain
VAR
	nSource: INT;
	nStartTimeInSeconds: UDINT ;
	nTime: UDINT;
	tempSecondsToAddWhilePause: INT;
	SecondsToAddWhilePause: INT;
	RemainingTime: UDINT;
	fb_FTRIG: R_TRIG;
	bStartCommand: BOOL;
	CLK: INT;
	Q: INT;
	b: BOOL;
	bN2PurgeBlockEnded: BOOL;
	fbSelection : FBSelection;
	

END_VAR

VAR_INPUT
	nCurrentBlock: INT;
	sSourceName: STRING;
END_VAR

fbSelection.TargetConverter(sTargetName:= sSourceName, TargetConverter_output => nSource); 


IF (RecipeTags.bStartTimeEnable[nCurrentBlock]=FALSE) THEN
	RecipeTags.Recipe.Blocks[nCurrentBlock].Properties.sStartTime:=MAIN.sConcatenatedHourMinuteString;
	nStartTimeInSeconds := STRING_TO_UDINT(MAIN.sCurrentSecond);
	RecipeTags.bStartTimeEnable[nCurrentBlock] :=  TRUE;
END_IF



IF RecipeTags.Recipe.Blocks[nCurrentBlock].Properties.sIntervalType = 'S' THEN
	nTime := DINT_TO_UDINT(RecipeTags.Recipe.Blocks[nCurrentBlock].Properties.nInterval);
ELSIF RecipeTags.Recipe.Blocks[nCurrentBlock].Properties.sIntervalType = 'M' THEN
	nTime := DINT_TO_UDINT(RecipeTags.Recipe.Blocks[nCurrentBlock].Properties.nInterval * 60);
ELSIF RecipeTags.Recipe.Blocks[nCurrentBlock].Properties.sIntervalType = 'H' THEN
	nTime := DINT_TO_UDINT(RecipeTags.Recipe.Blocks[nCurrentBlock].Properties.nInterval * 3600);
END_IF


IF RecipeTags.enWaitPause[nCurrentBlock] THEN
	tempSecondsToAddWhilePause := tempSecondsToAddWhilePause + 1;
	SecondsToAddWhilePause := tempSecondsToAddWhilePause; 
ELSE
	tempSecondsToAddWhilePause := 0;
END_IF

IF NOT(RecipeTags.bPauseRecipe) THEN
		RecipeTags.enWaitPause[nCurrentBlock] := FALSE;
		RecipeTags.bBlockStart[nCurrentBlock] := TRUE;
		RemainingTime := nTime- nStartTimeInSeconds-STRING_TO_UDINT(MAIN.sCurrentSecond);
ELSE
		RecipeTags.bBlockStart[nCurrentBlock] := FALSE;
		RecipeTags.enWaitPause[nCurrentBlock] := TRUE;
END_IF

IF  (nTime + nStartTimeInSeconds + DINT_TO_UDINT(TRUNC(SecondsToAddWhilePause/100))) <= (STRING_TO_UDINT(MAIN.sCurrentSecond)) AND RecipeTags.bSkipDrain THEN
	RecipeTags.Recipe.Blocks[nCurrentBlock].Properties.bStopCommand := TRUE;
	RecipeTags.Recipe.Blocks[nCurrentBlock].Properties.sEndTime:=MAIN.sConcatenatedHourMinuteString;
	RecipeTags.bBlockStart[nCurrentBlock] := FALSE;
	RecipeTags.bBlockEnd[nCurrentBlock] := TRUE;
	RecipeTags.bDrainStatus := FALSE;
	RecipeTags.bSkipDrain := FALSE;

ELSIF RecipeTags.bSkipDrain THEN
	RecipeTags.Recipe.Blocks[nCurrentBlock].Properties.bStopCommand := TRUE;
	RecipeTags.Recipe.Blocks[nCurrentBlock].Properties.sEndTime:=MAIN.sConcatenatedHourMinuteString;
	RecipeTags.bBlockStart[nCurrentBlock] := FALSE;
	RecipeTags.bBlockEnd[nCurrentBlock] := TRUE;
	RecipeTags.bDrainStatus := FALSE;
	RecipeTags.bSkipDrain := FALSE;
ELSE
	RecipeTags.bBlockEnd[nCurrentBlock] := FALSE;
END_IF

IF RecipeTags.bBlockStart[nCurrentBlock] THEN
	RecipeTags.bDrainStatus := TRUE;
	IF (nSource>=0 AND nSource<5) OR (nSource>6 AND nSource<=8) THEN
		IO.Vessels[nSource].Valves[0].bStart := TRUE;
	END_IF
	IF nSource=5 OR nSource=6 THEN
		IO.Vessels[nSource].Valves[6].bStart := TRUE;
		IO.Vessels[nSource].Valves[0].bStart := TRUE;
	END_IF
	//MVA drain
	IF nSource=9 AND nSource<10 THEN
		IO.Reactors[nSource-9].Valves[5].bStart := TRUE;
		IO.Reactors[nSource-9].Valves[0].bStart := TRUE;
		IO.Reactors[nSource-9].Valves[2].bStart := TRUE;
	END_IF
	//RV Drain
	IF nSource=10 OR nSource=11 THEN
		IO.Reactors[nSource-9].Valves[2].bStart := TRUE;
		IO.Reactors[nSource-9].Valves[0].bStart := TRUE;

	END_IF
ELSE
	IF (nSource>=0 AND nSource<5) OR (nSource>6 AND nSource<=8) THEN
		IO.Vessels[nSource].Valves[0].bStart := FALSE;
	END_IF
	IF nSource<9 THEN
		IO.Vessels[nSource].Valves[6].bStart := FALSE;
		IO.Vessels[nSource].Valves[0].bStart := false;

	END_IF
	//MVA drain
	IF nSource=9 AND nSource<10 THEN
		IO.Reactors[nSource-9].Valves[5].bStart := FALSE;
		IO.Reactors[nSource-9].Valves[0].bStart := FALSE;
		IO.Reactors[nSource-9].Valves[2].bStart := FALSE;
	END_IF
	IF nSource=10 OR nSource=11 THEN
		IO.Reactors[nSource-9].Valves[2].bStart := FALSE;
		IO.Reactors[nSource-9].Valves[0].bStart := FALSE;

	END_IF
END_IF

fb_FTRIG(CLK:=RecipeTags.bBlockEnd[nCurrentBlock], Q=> );
IF fb_FTRIG.Q AND RecipeTags.Recipe.Blocks[nCurrentBlock].Name = 'Drain' THEN
	RecipeTags.bSkipDrain := FALSE;
	RecipeTags.bDrainStatus := FALSE;
	RecipeTags.bBlockEnd[nCurrentBlock] := FALSE;
	RecipeTags.bStartTimeEnable[nCurrentBlock] :=  FALSE;
	SecondsToAddWhilePause := 0;
	nTime := 0;
	nStartTimeInSeconds := 0;
	RecipeTags.Recipe.Blocks[nCurrentBlock].Properties.sEndTime:=MAIN.sConcatenatedHourMinuteString;
	RecipeTags.Recipe.Blocks[nCurrentBlock].Properties.bStopCommand := TRUE;
END_IF

END_PROGRAM

// ---- RecipeControl/RecipeBlocks/N2Purge/N2Purge.TcPOU
PROGRAM N2Purge
VAR
	nSource: INT;
	nStartTimeInSeconds: UDINT ;
	nTime: UDINT;
	tempSecondsToAddWhilePause: DINT;
	SecondsToAddWhilePause: DINT;
	RemainingTime: UDINT;
	fb_FTRIG: R_TRIG;
	bStartCommand: BOOL;
	CLK: INT;
	Q: INT;
	b: BOOL;
	bN2PurgeBlockEnded: BOOL;
	fbSelection : FBSelection;
	

END_VAR

VAR_INPUT
	nCurrentBlock: INT;
	sSourceName: STRING;
END_VAR

fbSelection.TargetConverter(sTargetName:= sSourceName, TargetConverter_output => nSource); 

IF RecipeTags.Recipe.Blocks[nCurrentBlock].Properties.sStartTime = '' THEN
	RecipeTags.StaredTimeForRecipeBanner := MAIN.concatenatedHourMinuteString;
END_IF
IF (RecipeTags.bStartTimeEnable[nCurrentBlock]=FALSE) THEN
//	RecipeControl.StaredTimeForRecipeBanner := MAIN.concatenatedHourMinuteString;
	RecipeTags.Recipe.Blocks[nCurrentBlock].Properties.sStartTime:=MAIN.sConcatenatedHourMinuteString;
	nStartTimeInSeconds := STRING_TO_UDINT(MAIN.sCurrentSecond);
	RecipeTags.bStartTimeEnable[nCurrentBlock] :=  TRUE;
END_IF



IF RecipeTags.Recipe.Blocks[nCurrentBlock].Properties.sIntervalType = 'S' THEN
	nTime := DINT_TO_UDINT(RecipeTags.Recipe.Blocks[nCurrentBlock].Properties.nInterval);
ELSIF RecipeTags.Recipe.Blocks[nCurrentBlock].Properties.sIntervalType = 'M' THEN
	nTime := DINT_TO_UDINT(RecipeTags.Recipe.Blocks[nCurrentBlock].Properties.nInterval * 60);
ELSIF RecipeTags.Recipe.Blocks[nCurrentBlock].Properties.sIntervalType = 'H' THEN
	nTime := DINT_TO_UDINT(RecipeTags.Recipe.Blocks[nCurrentBlock].Properties.nInterval * 3600);
END_IF



IF RecipeTags.enWaitPause[nCurrentBlock] THEN
	tempSecondsToAddWhilePause := tempSecondsToAddWhilePause + 1;
	SecondsToAddWhilePause := tempSecondsToAddWhilePause; 
ELSE
	tempSecondsToAddWhilePause := 0;
	SecondsToAddWhilePause :=0;

END_IF

IF NOT(RecipeTags.bPauseRecipe) THEN
		RecipeTags.enWaitPause[nCurrentBlock] := FALSE;
		RecipeTags.bBlockStart[nCurrentBlock] := TRUE;
		RemainingTime := nTime- nStartTimeInSeconds-STRING_TO_UDINT(MAIN.sCurrentSecond);
ELSE
		RecipeTags.bBlockStart[nCurrentBlock] := FALSE;
		RecipeTags.enWaitPause[nCurrentBlock] := TRUE;
END_IF


IF  (nTime + nStartTimeInSeconds + DINT_TO_UDINT(TRUNC(SecondsToAddWhilePause/100))) <= (STRING_TO_UDINT(MAIN.sCurrentSecond)) THEN
	RecipeTags.Recipe.Blocks[nCurrentBlock].Properties.bStopCommand := TRUE;
	RecipeTags.Recipe.Blocks[nCurrentBlock].Properties.sEndTime:=MAIN.sConcatenatedHourMinuteString;
	RecipeTags.bBlockStart[nCurrentBlock] := FALSE;
	RecipeTags.bBlockEnd[nCurrentBlock] := TRUE;
ELSE
	RecipeTags.bBlockEnd[nCurrentBlock] := FALSE;

END_IF

IF RecipeTags.bBlockStart[nCurrentBlock] THEN
	IF nSource<9 THEN
		IO.Vessels[nSource].Valves[1].bStart := TRUE;
	END_IF
	IF nSource>=9 AND nSource<=11 THEN
		IO.Reactors[nSource-9].Valves[1].bStart := TRUE;
	END_IF
ELSE
	IF nSource<9 THEN
		IO.Vessels[nSource].Valves[1].bStart := FALSE;
	END_IF
	IF nSource>=9 AND nSource<=11 THEN
		IO.Reactors[nSource-9].Valves[1].bStart := FALSE;
	end_if
END_IF

fb_FTRIG(CLK:=RecipeTags.bBlockEnd[nCurrentBlock], Q=> );
IF fb_FTRIG.Q AND RecipeTags.Recipe.Blocks[nCurrentBlock].Name = 'N2Purge' THEN
	RecipeTags.Recipe.Blocks[nCurrentBlock].Properties.sEndTime:=MAIN.sConcatenatedHourMinuteString;
	RecipeTags.Recipe.Blocks[nCurrentBlock].Properties.bStopCommand := TRUE;
	RecipeTags.bBlockEnd[nCurrentBlock] := FALSE;
	RecipeTags.bStartTimeEnable[nCurrentBlock] :=  FALSE;

END_IF

END_PROGRAM

// ---- RecipeControl/ClearRecipe.TcPOU
PROGRAM ClearRecipe
VAR
	i: INT;
	j: INT;
END_VAR

//Manual Logic for Reactors.Valves
	
FOR i:=0 TO 1 DO
	FOR j :=0 TO 7 DO
		IO.Reactors[i].Valves[j].bStart :=	FALSE;
	END_FOR
END_FOR
	
	//Manual Logic for Reactors.Pumps
	
FOR i:=0 TO 1 DO
	FOR j :=0 TO 1 DO
		IO.Reactors[i].Pumps[j].bStart :=FALSE;
	END_FOR
END_FOR

FOR i := 0 TO 699 DO
	RecipeTags.Recipe.Blocks[i].Properties.bBlockStarted := FALSE;
	RecipeTags.Recipe.Blocks[i].Properties.bStartCommand := FALSE;
	RecipeTags.Recipe.Blocks[i].Properties.bBlockEnded := FALSE;
	RecipeTags.Recipe.Blocks[i].Properties.bStopCommand := FALSE;
	RecipeTags.Recipe.Blocks[i].Properties.bModeSelection := FALSE;
	RecipeTags.Recipe.Blocks[i].Properties.sStartTime := '';
	RecipeTags.Recipe.Blocks[i].Properties.sEndTime := '';
	
	RecipeTags.SlaveRecipe.Blocks[i].Properties.bBlockStarted := FALSE;
	RecipeTags.SlaveRecipe.Blocks[i].Properties.bStartCommand := FALSE;
	RecipeTags.SlaveRecipe.Blocks[i].Properties.bBlockEnded := FALSE;
	RecipeTags.SlaveRecipe.Blocks[i].Properties.bStopCommand := FALSE;
	RecipeTags.SlaveRecipe.Blocks[i].Properties.bModeSelection := FALSE;
	RecipeTags.SlaveRecipe.Blocks[i].Properties.sStartTime := '';
	RecipeTags.SlaveRecipe.Blocks[i].Properties.sEndTime := '';
	
	RecipeTags.bBlockStart[i] := FALSE;
	RecipeTags.enWaitPause[i] := FALSE;
	RecipeTags.bBlockEnd[i] := FALSE;
	RecipeTags.bStartTimeEnable[i] := FALSE;

END_FOR


FOR i := 0 TO 2 DO
	IO.Reactors[i].VFD.bStart := FALSE;
	IO.Reactors[i].VFD.nRPMSetPointScaled := 0; 
END_FOR

FOR i:=0 TO 8 DO
	FOR j :=0 TO 7 DO
		IO.Vessels[i].Valves[j].bStart := FALSE;
	END_FOR
END_FOR
	
	//Manual Logic for Vessels.Pumps
	
FOR i:=0 TO 8 DO
	FOR j :=0 TO 1 DO
		IO.Vessels[i].Pumps[j].bStart :=FALSE;
	END_FOR
END_FOR

RecipeTags.bDrainStatus := FALSE;
RecipeTags.bSkipDrain := FALSE;
RecipeTags.bPauseRecipe := FALSE;
RecipeTags.bTransferStartTime	 := FALSE;

END_PROGRAM

// ---- POUs/AnalogScaling_1.TcPOU
PROGRAM AnalogScaling_1
VAR_INPUT

END_VAR
VAR
	fbScaling: ARRAY[0..15] OF FB_Scaling;
	i: INT;
	tempTagForChangingDec : ARRAY[0..15] OF REAL;
	
	fbTON :TON;
	fbTONTrig : TON;
	
	fbStirControl : FBStirControl;
	iStirControl : IStirControl;

END_VAR

iStirControl := fbStirControl;

IF iStirControl <> 0 THEN
	iStirControl := iStirControl;
END_IF
	



//=========================================================
//  Scaling

//FOR i:=0 TO 1 DO
//	fbScaling[0](
//		nRawInputValue:= IO.Reactors[i].Temperature.RawValue, 
//		nInputLowerLimit:= IO.Reactors[i].Temperature.RawLowLimit, 
//		nInputHigherLimit:= IO.Reactors[i].Temperature.RawHighLimit, 
//		nOutputLowerLimit:= IO.Reactors[i].Temperature.ScaledLowLimit, 
//		nOutputHigherLimit:= IO.Reactors[i].Temperature.ScaledHighLimit, 
//		nScaledValueF=> tempTagForChangingDec[i], 
//		nScaledValueD=> );
	
//	IO.Reactors[i].Temperature.ScaledValue := INT_TO_LREAL(LREAL_TO_INT(tempTagForChangingDec[i]*100))/100;
	
//	fbScaling[1](
//		nRawInputValue:= IO.Reactors[i].Pressure.RawValue, 
//		nInputLowerLimit:= IO.Reactors[i].Pressure.RawLowLimit, 
//		nInputHigherLimit:= IO.Reactors[i].Pressure.RawHighLimit, 
//		nOutputLowerLimit:= IO.Reactors[i].Pressure.ScaledLowLimit, 
//		nOutputHigherLimit:= IO.Reactors[i].Pressure.ScaledHighLimit, 
//		nScaledValueF=> tempTagForChangingDec[i], 
//		nScaledValueD=> );
	
//	IO.Reactors[i].Pressure.ScaledValue := INT_TO_LREAL(LREAL_TO_INT(tempTagForChangingDec[i]*100))/100;
	
//	fbScaling[2](
//		nRawInputValue:= IO.Reactors[i].Level.RawValue, 
//		nInputLowerLimit:= IO.Reactors[i].Level.RawLowLimit, 
//		nInputHigherLimit:= IO.Reactors[i].Level.RawHighLimit, 
//		nOutputLowerLimit:= IO.Reactors[i].Level.ScaledLowLimit, 
//		nOutputHigherLimit:= IO.Reactors[i].Level.ScaledHighLimit, 
//		nScaledValueF=> tempTagForChangingDec[i], 
//		nScaledValueD=> );
	
//	IO.Reactors[i].Level.ScaledValue := INT_TO_LREAL(LREAL_TO_INT(tempTagForChangingDec[i]*100))/100;	
		
//	fbScaling[3](
//		nRawInputValue:= IO.Reactors[i].VFD.nRPMFeedBackRaw, 
//		nInputLowerLimit:= 0, 
//		nInputHigherLimit:= 32767, 
//		nOutputLowerLimit:= 0, 
//		nOutputHigherLimit:= 200, 
//		nScaledValueF=> tempTagForChangingDec[3], 
//		nScaledValueD=> );
		
//	IO.Reactors[i].VFD.nRPMFeedBackScaled := INT_TO_LREAL(LREAL_TO_INT(tempTagForChangingDec[i]));		
		
//	fbScaling[4](
//		nRawInputValue:= REAL_TO_INT(IO.Reactors[i].VFD.nRPMSetPointScaled), 
//		nInputLowerLimit:= 0, 
//		nInputHigherLimit:= 200, 
//		nOutputLowerLimit:= 6553, 
//		nOutputHigherLimit:= 32767, 
//		nScaledValueF=> , 
//		nScaledValueD=> );
	
//	IO.Reactors[i].VFD.nRPMSetPointRaw := LREAL_TO_INT(fbScaling[4].nScaledValueF);
	
//END_FOR

fbScaling[0](
		nRawInputValue:= IO.Reactors[0].Temperature.RawValue, 
		nInputLowerLimit:= IO.Reactors[0].Temperature.RawLowLimit, 
		nInputHigherLimit:= IO.Reactors[0].Temperature.RawHighLimit, 
		nOutputLowerLimit:= IO.Reactors[0].Temperature.ScaledLowLimit, 
		nOutputHigherLimit:= IO.Reactors[0].Temperature.ScaledHighLimit, 
		nScaledValueF=> tempTagForChangingDec[0], 
		nScaledValueD=> );
	
	IO.Reactors[0].Temperature.ScaledValue := INT_TO_LREAL(LREAL_TO_INT(tempTagForChangingDec[0]*100))/100;

fbScaling[1](
		nRawInputValue:= IO.Reactors[1].Temperature.RawValue, 
		nInputLowerLimit:= IO.Reactors[1].Temperature.RawLowLimit, 
		nInputHigherLimit:= IO.Reactors[1].Temperature.RawHighLimit, 
		nOutputLowerLimit:= IO.Reactors[1].Temperature.ScaledLowLimit, 
		nOutputHigherLimit:= IO.Reactors[1].Temperature.ScaledHighLimit, 
		nScaledValueF=> tempTagForChangingDec[1], 
		nScaledValueD=> );
	
	IO.Reactors[1].Temperature.ScaledValue := INT_TO_LREAL(LREAL_TO_INT(tempTagForChangingDec[1]*100))/100;

fbScaling[2](
		nRawInputValue:= IO.Reactors[2].Temperature.RawValue, 
		nInputLowerLimit:= IO.Reactors[2].Temperature.RawLowLimit, 
		nInputHigherLimit:= IO.Reactors[2].Temperature.RawHighLimit, 
		nOutputLowerLimit:= IO.Reactors[2].Temperature.ScaledLowLimit, 
		nOutputHigherLimit:= IO.Reactors[2].Temperature.ScaledHighLimit, 
		nScaledValueF=> tempTagForChangingDec[2], 
		nScaledValueD=> );
	
	IO.Reactors[2].Temperature.ScaledValue := INT_TO_LREAL(LREAL_TO_INT(tempTagForChangingDec[2]*100))/100;
	
fbScaling[3](
		nRawInputValue:= IO.Reactors[0].Pressure.RawValue, 
		nInputLowerLimit:= IO.Reactors[0].Pressure.RawLowLimit, 
		nInputHigherLimit:= IO.Reactors[0].Pressure.RawHighLimit, 
		nOutputLowerLimit:= IO.Reactors[0].Pressure.ScaledLowLimit, 
		nOutputHigherLimit:= IO.Reactors[0].Pressure.ScaledHighLimit, 
		nScaledValueF=> tempTagForChangingDec[3], 
		nScaledValueD=> );
	
	IO.Reactors[0].Pressure.ScaledValue := INT_TO_LREAL(LREAL_TO_INT(tempTagForChangingDec[3]*100))/100;

fbScaling[4](
		nRawInputValue:= IO.Reactors[1].Pressure.RawValue, 
		nInputLowerLimit:= IO.Reactors[1].Pressure.RawLowLimit, 
		nInputHigherLimit:= IO.Reactors[1].Pressure.RawHighLimit, 
		nOutputLowerLimit:= IO.Reactors[1].Pressure.ScaledLowLimit, 
		nOutputHigherLimit:= IO.Reactors[1].Pressure.ScaledHighLimit, 
		nScaledValueF=> tempTagForChangingDec[4], 
		nScaledValueD=> );
	
	IO.Reactors[1].Pressure.ScaledValue := INT_TO_LREAL(LREAL_TO_INT(tempTagForChangingDec[4]*100))/100;

fbScaling[5](
		nRawInputValue:= IO.Reactors[2].Pressure.RawValue, 
		nInputLowerLimit:= IO.Reactors[2].Pressure.RawLowLimit, 
		nInputHigherLimit:= IO.Reactors[2].Pressure.RawHighLimit, 
		nOutputLowerLimit:= IO.Reactors[2].Pressure.ScaledLowLimit, 
		nOutputHigherLimit:= IO.Reactors[2].Pressure.ScaledHighLimit, 
		nScaledValueF=> tempTagForChangingDec[5], 
		nScaledValueD=> );
	
	IO.Reactors[2].Pressure.ScaledValue := INT_TO_LREAL(LREAL_TO_INT(tempTagForChangingDec[5]*100))/100;
	
fbScaling[6](
		nRawInputValue:= IO.Reactors[0].Level.RawValue, 
		nInputLowerLimit:= 15780, 
		nInputHigherLimit:= 27500, 
		nOutputLowerLimit:= IO.Reactors[0].Level.ScaledLowLimit, 
		nOutputHigherLimit:= IO.Reactors[0].Level.ScaledHighLimit, 
		nScaledValueF=> tempTagForChangingDec[6], 
		nScaledValueD=> );
		
		IF (tempTagForChangingDec[6] < 0) THEN
			IO.Reactors[0].Level.ScaledValue := 0;
		ELSIF (tempTagForChangingDec[6] > 100) THEN
			IO.Reactors[0].Level.ScaledValue := 100;
		ELSE
			IO.Reactors[0].Level.ScaledValue := INT_TO_LREAL(LREAL_TO_INT(tempTagForChangingDec[6]*100))/100;	
		END_IF
	

fbScaling[7](
		nRawInputValue:= IO.Reactors[1].Level.RawValue, 
		nInputLowerLimit:= 2500, 
		nInputHigherLimit:= 20000, 
		nOutputLowerLimit:= IO.Reactors[1].Level.ScaledLowLimit, 
		nOutputHigherLimit:= IO.Reactors[1].Level.ScaledHighLimit, 
		nScaledValueF=> tempTagForChangingDec[7], 
		nScaledValueD=> );
		IF (tempTagForChangingDec[7] < 0) THEN
			IO.Reactors[1].Level.ScaledValue := 0;
		ELSIF (tempTagForChangingDec[7] > 100) THEN
			IO.Reactors[1].Level.ScaledValue := 100;
		ELSE
			IO.Reactors[1].Level.ScaledValue := INT_TO_LREAL(LREAL_TO_INT(tempTagForChangingDec[7]*100))/100;	
		END_IF
	
	
fbScaling[8](
		nRawInputValue:= IO.Reactors[2].Level.RawValue, 
		nInputLowerLimit:= 0, 
		nInputHigherLimit:= 23120, 
		nOutputLowerLimit:= IO.Reactors[2].Level.ScaledLowLimit, 
		nOutputHigherLimit:= IO.Reactors[2].Level.ScaledHighLimit, 
		nScaledValueF=> tempTagForChangingDec[8], 
		nScaledValueD=> );
	
	IO.Reactors[2].Level.ScaledValue := INT_TO_LREAL(LREAL_TO_INT(tempTagForChangingDec[8]*100))/100;	
		
	fbScaling[9](
		nRawInputValue:= IO.Reactors[0].VFD.nRPMFeedBackRaw, 
		nInputLowerLimit:= 0, 
		nInputHigherLimit:= 32767, 
		nOutputLowerLimit:= 0, 
		nOutputHigherLimit:= 200, 
		nScaledValueF=> tempTagForChangingDec[9], 
		nScaledValueD=> );
		
		IF (INT_TO_LREAL(LREAL_TO_INT(tempTagForChangingDec[9]))) < 5 THEN
			IO.Reactors[0].VFD.nRPMFeedBackScaled := 0;
		ELSE
			IO.Reactors[0].VFD.nRPMFeedBackScaled := INT_TO_LREAL(LREAL_TO_INT(tempTagForChangingDec[9]));		
		END_IF
	
fbScaling[10](
		nRawInputValue:= IO.Reactors[1].VFD.nRPMFeedBackRaw, 
		nInputLowerLimit:= 0, 
		nInputHigherLimit:= 32767, 
		nOutputLowerLimit:= 0, 
		nOutputHigherLimit:= 200, 
		nScaledValueF=> tempTagForChangingDec[10], 
		nScaledValueD=> );
	
		IF (INT_TO_LREAL(LREAL_TO_INT(tempTagForChangingDec[10]))) < 5 THEN
			IO.Reactors[1].VFD.nRPMFeedBackScaled := 0;
		ELSE
			IO.Reactors[1].VFD.nRPMFeedBackScaled := INT_TO_LREAL(LREAL_TO_INT(tempTagForChangingDec[10]));		
		END_IF
	
		
	
fbScaling[11](
		nRawInputValue:= IO.Reactors[2].VFD.nRPMFeedBackRaw, 
		nInputLowerLimit:= 0, 
		nInputHigherLimit:= 32767, 
		nOutputLowerLimit:= 0, 
		nOutputHigherLimit:= 200, 
		nScaledValueF=> tempTagForChangingDec[11], 
		nScaledValueD=> );
		IF (INT_TO_LREAL(LREAL_TO_INT(tempTagForChangingDec[11]))) < 5 THEN
			IO.Reactors[2].VFD.nRPMFeedBackScaled := 0;
		ELSE
			IO.Reactors[2].VFD.nRPMFeedBackScaled := INT_TO_LREAL(LREAL_TO_INT(tempTagForChangingDec[11]));		
		END_IF
		
 //VFDSetpointOutput => fb_scaling[0].nRawInputValue);
iStirControl.StirControl(i:=0);
fbScaling[12](
		nRawInputValue:= LREAL_TO_INT(iStirControl.pSetpoint), 
		nInputLowerLimit:= 0, 
		nInputHigherLimit:= 200, 
		nOutputLowerLimit:= 6553, 
		nOutputHigherLimit:= 32767, 
		nScaledValueF=> tempTagForChangingDec[12], 
		nScaledValueD=> );
		IO.Reactors[0].VFD.nRPMSetPointRaw := LREAL_TO_INT(tempTagForChangingDec[12]);		

iStirControl.StirControl(i:=1);
fbScaling[13](
		nRawInputValue:= LREAL_TO_INT(iStirControl.pSetpoint), 
		nInputLowerLimit:= 0, 
		nInputHigherLimit:= 200, 
		nOutputLowerLimit:= 6553, 
		nOutputHigherLimit:= 32767, 
		nScaledValueF=> tempTagForChangingDec[13], 
		nScaledValueD=> );
		IO.Reactors[1].VFD.nRPMSetPointRaw := LREAL_TO_INT(tempTagForChangingDec[13]);		
	
iStirControl.StirControl(i:=2);
fbScaling[14](
		nRawInputValue:= LREAL_TO_INT(iStirControl.pSetpoint), 
		nInputLowerLimit:= 0, 
		nInputHigherLimit:= 200, 
		nOutputLowerLimit:= 6553, 
		nOutputHigherLimit:= 32767, 
		nScaledValueF=> tempTagForChangingDec[14], 
		nScaledValueD=> );
		IO.Reactors[2].VFD.nRPMSetPointRaw := LREAL_TO_INT(tempTagForChangingDec[14]);		
		
fbScaling[15](
		nRawInputValue:= IO.PhysicalIO.JacketTemperature, 
		nInputLowerLimit:= 0, 
		nInputHigherLimit:= 32767, 
		nOutputLowerLimit:= 0, 
		nOutputHigherLimit:= 200, 
		nScaledValueF=> tempTagForChangingDec[15], 
		nScaledValueD=> );
		IO.JacketTemperature := INT_TO_LREAL(LREAL_TO_INT(tempTagForChangingDec[15]*100))/100;

END_PROGRAM

// ---- Helpers/FB_Scaling.TcPOU
FUNCTION_BLOCK FB_Scaling
VAR_INPUT
	nRawInputValue			: INT;
	nInputLowerLimit		: INT;
	nInputHigherLimit		: DINT;
	nOutputLowerLimit		: LREAL;
	nOutputHigherLimit		: LREAL;
END_VAR
VAR_OUTPUT 
		nScaledValueF		: LREAL;
	    nScaledValueD		: INT;
END_VAR
VAR
	 nGain		: REAL;
	Temp: STRING(510);
END_VAR

// Scaling Calculations //

	IF	nRawInputValue	<	0	THEN
		nRawInputValue	:=	0;
	END_IF


	IF	 ((nInputHigherLimit - nInputLowerLimit)	<= 0)	THEN
//		 ((nOutputHigherLimit  - nOutputLowerLimit)	<= 0)	THEN
		nGain	:=	0;
	ELSE
//				nGain:=(((nRawInputValue - nInputLowerLimit) / (nInputHigherLimit - nInputLowerLimit)) * (nOutputHigherLimit  - nOutputLowerLimit)) + nOutputLowerLimit;
		nGain:=(nRawInputValue - nInputLowerLimit)*((nOutputHigherLimit - nOutputLowerLimit) / (nInputHigherLimit - nInputLowerLimit)) + nOutputLowerLimit;
	END_IF


		Temp	:=	LREAL_TO_FMTSTR( nGain, 1, TRUE );
		
		nScaledValueF	:=	STRING_TO_REAL(Temp);
		nScaledValueD	:=	REAL_TO_INT(nGain);

END_FUNCTION_BLOCK

// ---- POUs/Modbus.TcPOU
PROGRAM Modbus
VAR
	fbModbusRtuMaster_PcCOM:ModbusRtuMaster_PcCOM;
	ChillerRead : ARRAY[0..10] OF WORD;
	ChillerWrite : ARRAY[0..10] OF WORD;

	bWrite: BOOL;
	bRead: BOOL;
	
	fbTON :TON;
	fbTONTrig : TON;
END_VAR

fbTON(IN:=NOT(fbTONTrig.Q), PT:= T#1S);
fbTONTrig(IN:=fbTON.Q, PT:= T#1s);


fbModbusRtuMaster_PcCOM.ReadRegs(
	UnitID:= 01, 
	Quantity:= 7, 
	MBAddr:= 16#0
, 
	cbLength:= SIZEOF(ChillerRead), 
	pMemoryAddr:= ADR(ChillerRead), 
	Execute:= fbTON.Q, 
	Timeout:= T#5S);
	
IO.ChillerTemperature := WORD_TO_REAL(ChillerRead[5]);
ChillerWrite[0] := REAL_TO_WORD(IO.ChillerTempSetpoint);	
	
fbModbusRtuMaster_PcCOM.WriteRegs(
	UnitID:= 01, 
	Quantity:= 1, 
	MBAddr:= 16#8, 
	cbLength:= SIZEOF(ChillerWrite), 
	pMemoryAddr:= ADR(ChillerWrite), 
	Execute:= NOT(fbTON.Q), 
	Timeout:= T#5S);

END_PROGRAM

// ---- AnalogScaling.TcPOU
PROGRAM AnalogScaling
VAR
	fbScaling: FB_Scaling;
	i: INT;
END_VAR

//=========================================================
// RV  Scaling

FOR i:=0 TO 2 DO
	fbScaling(
		nRawInputValue:= IO.Reactors[i].Temperature.RawValue, 
		nInputLowerLimit:= IO.Reactors[i].Temperature.RawLowLimit, 
		nInputHigherLimit:= IO.Reactors[i].Temperature.RawHighLimit, 
		nOutputLowerLimit:= IO.Reactors[i].Temperature.ScaledLowLimit, 
		nOutputHigherLimit:= IO.Reactors[i].Temperature.ScaledHighLimit, 
		nScaledValueF=> IO.Reactors[i].Temperature.ScaledValue, 
		nScaledValueD=> );
	
	fbScaling(
		nRawInputValue:= IO.Reactors[i].Pressure.RawValue, 
		nInputLowerLimit:= IO.Reactors[i].Pressure.RawLowLimit, 
		nInputHigherLimit:= IO.Reactors[i].Pressure.RawHighLimit, 
		nOutputLowerLimit:= IO.Reactors[i].Pressure.ScaledLowLimit, 
		nOutputHigherLimit:= IO.Reactors[i].Pressure.ScaledHighLimit, 
		nScaledValueF=> IO.Reactors[i].Pressure.ScaledValue, 
		nScaledValueD=> );
	
	fbScaling(
		nRawInputValue:= IO.Reactors[i].Level.RawValue, 
		nInputLowerLimit:= IO.Reactors[i].Level.RawLowLimit, 
		nInputHigherLimit:= IO.Reactors[i].Level.RawHighLimit, 
		nOutputLowerLimit:= IO.Reactors[i].Level.ScaledLowLimit, 
		nOutputHigherLimit:= IO.Reactors[i].Level.ScaledHighLimit, 
		nScaledValueF=> IO.Reactors[i].Level.ScaledValue, 
		nScaledValueD=> );

END_FOR

END_PROGRAM

// ---- Manualmplementation/FB_ManualImplementation_1.TcPOU
FUNCTION_BLOCK FB_ManualImplementation_1 IMPLEMENTS  I_ManualImplementation
VAR_INPUT
		i_ManualControl : ARRAY[0..10,0..10] OF I_ManualControl;
END_VAR
VAR_OUTPUT
END_VAR
VAR
	i: INT;
	j: INT;
	k: INT;
	k_1: INT;
END_VAR

//=========================================================
// Instantiation Logic


	FOR k:=0 TO 10 DO
		FOR k_1 := 0 TO 10 DO
			IF i_ManualControl[k, k_1] <> 0 THEN
			THIS^.i_ManualControl[k, k_1] := i_ManualControl[k, k_1];
		END_IF	
		END_FOR
		
	END_FOR


//=========================================================
// Count Declaration Logic

	

//=========================================================
// Manual Logic
	
	//Manual Logic for Vessels.Valves
	
	FOR i:=0 TO 8 DO
		FOR j :=0 TO 7 DO
			IO.Vessels[i].Valves[j].Output :=i_ManualControl[i, j].
				M_RunValve(IO.Vessels[i].Valves[j].bStart);
		END_FOR
	END_FOR
	
	//Manual Logic for Vessels.Pumps
	
	FOR i:=0 TO 8 DO
		FOR j :=0 TO 1 DO
			IO.Vessels[i].Pumps[j].nPulse := 4;
			IO.Vessels[i].Pumps[j].Output :=i_ManualControl[i,j].
				M_RunPump(IO.Vessels[i].Pumps[j].bStart,IO.Vessels[i].Pumps[j].nPulse);
		END_FOR
	END_FOR
	
	//Manual Logic for Reactors.Valves
	
	FOR i:=0 TO 1 DO
		FOR j :=0 TO 7 DO
			IO.Reactors[i].Valves[j].Output :=i_ManualControl[9+i,j].
				M_RunValve(IO.Reactors[i].Valves[j].bStart);
		END_FOR
	END_FOR
	
	//Manual Logic for Reactors.Pumps
	
	FOR i:=0 TO 1 DO
		FOR j :=0 TO 1 DO
			IO.Reactors[i].Pumps[j].nPulse := 4;
			IO.Reactors[i].Pumps[j].Output :=i_ManualControl[9+i,j].
				M_RunPump(IO.Reactors[i].Pumps[j].bStart,IO.Reactors[i].Pumps[j].nPulse);
		END_FOR
	END_FOR

PROPERTY ipManualControl : ARRAY [0..10,0..10] OF I_ManualControl
GET
ipManualControl	:= i_ManualControl;
END_GET
END_PROPERTY

END_FUNCTION_BLOCK

// ---- Manualmplementation/ManualControl/FB_ManualControl_1.TcPOU
FUNCTION_BLOCK FB_ManualControl_1 IMPLEMENTS  I_ManualControl
VAR_INPUT
END_VAR
VAR_OUTPUT
END_VAR
VAR
	TEMP_1 : BOOL;
	Counter : INT;
	TEMP : BOOL;

	
END_VAR

{warning 'add method implementation '}
METHOD M_RunPump : BOOL
VAR_INPUT
	bStart	: BOOL;
	NTimes : INT;

END_VAR
VAR
	
END_VAR

IF NTimes <> 0 THEN
	IF TRUE THEN
	Counter := Counter + 1;
	END_IF
	IF Counter >= (100/(2*NTimes)) THEN
		TEMP := TRUE;
	ELSE
		TEMP := FALSE;
	END_IF
	IF Counter >= (200/(2*NTimes)) THEN
		Counter := 0;
	END_IF
ELSE
	RETURN;
END_IF

IF bstart THEN
	M_RunPump := TEMP;
ELSE
	M_RunPump := FALSE;
END_IF
END_METHOD

